    |     m3 = multiply_matrix(m2, m1)
    |     rxryrz1 = convert_matrix_to_axang(m3)
    |     rx1 = rxryrz1[0]
    |     ry1 = rxryrz1[1]
    |     rz1 = rxryrz1[2]
    | 
    |     point1 = p[p1x, p1y, p1z, rx1, ry1, rz1]
    | 
    |     # get second point (right) (point2)
    |     # take the center point and move right the radius plus the cushions
    |     p2x = pcx + vecrx * radius + vecrx * cusharound + vecnx * -1 * cushout
    |     p2y = pcy + vecry * radius + vecry * cusharound + vecny * -1 * cushout
    |     p2z = pcz
    | 
    |     # find rxryrz2
    |     # first rotation is 90 degrees about the x- axis
    |     m1 = get_rotation_matrix_from_description("x", -1, 90 * pi / 180)
    |     # second rotation is About 135 degrees about the z+ axis. This calculation is heading1 – 45 degrees
    |     m2 = get_rotation_matrix_from_description("z", 1, heading1 - 45 * pi/180)
    |     # combine them by multiplying
    |     m3 = multiply_matrix(m2, m1)
    |     rxryrz2 = convert_matrix_to_axang(m3)
    |     rx2 = rxryrz2[0]
    |     ry2 = rxryrz2[1]
    |     rz2 = rxryrz2[2]
    | 
    |     point2 = p[p2x, p2y, p2z, rx2, ry2, rz2]
    | 
    |     # get the third point (bottom) (point3)
    |     p3x = pcx + vecnx * -1 * cushout
    |     p3y = pcy + vecny * -1 * cushout
    |     p3z = pcz - vecuz * radius - vecuz * cusharound
    | 
    |     # find rxryrz3
    |     # first rotation is 45 degrees about the y+ axis
    |     m1 = get_rotation_matrix_from_description("y", 1, 45 * pi / 180)
    |     # second rotation is About 180 degrees about the z+ axis. This calculation is heading1 degrees
    |     m2 = get_rotation_matrix_from_description("z", 1, heading1)
    |     # combine them by multiplying
    |     m3 = multiply_matrix(m2, m1)
    |     rxryrz3 = convert_matrix_to_axang(m3)
    |     rx3 = rxryrz3[0]
    |     ry3 = rxryrz3[1]
    |     rz3 = rxryrz3[2]
    | 
    |     point3 = p[p3x, p3y, p3z, rx3, ry3, rz3]
    | 
    |     # get the fourth point (left) (point4)
    |     p4x = pcx - vecrx * radius - vecrx * cusharound + vecnx * -1 * cushout
    |     p4y = pcy - vecry * radius - vecry * cusharound + vecny * -1 * cushout
    |     p4z = pcz
    | 
    |     # find rxryrz4
    |     # first rotation is 90 degrees about the x+ axis
    |     m1 = get_rotation_matrix_from_description("x", 1, 90 * pi / 180)
    |     # second rotation is heading1 + 45 degrees about the z+ axis. approx 225 degrees ccw
    |     m2 = get_rotation_matrix_from_description("z", 1, heading1 + 45 * pi/180)
    |     # combine them by multiplying
    |     m3 = multiply_matrix(m2, m1)
    |     rxryrz4 = convert_matrix_to_axang(m3)
    |     rx4 = rxryrz4[0]
    |     ry4 = rxryrz4[1]
    |     rz4 = rxryrz4[2]
    | 
    |     point4 = p[p4x, p4y, p4z, rx4, ry4, rz4]
    | 
    |     # return the points
    |     ret = struct(point1=point1, point2=point2, point3=point3, point4=point4)
    |     return ret
    | 
    | end
    | 
    | # this function calculates the points necessary for the fillet sleeve weld path.
    | # this assumes a vertical plane
    | def calculate_points_sleeve_fillet(struct1):
    |     # get the stuff from the struct
    |     pcenter = struct1[0]
    |     pcx = pcenter[0]
    |     pcy = pcenter[1]
    |     pcz = pcenter[2]
    |     planenormalvec = struct1[1]
    |     radius = struct1[2]
    |     heading1 = struct1[3]
    |     vecn = struct1[4]
    |     vecnx = vecn[0]
    |     vecny = vecn[1]
    |     vecr = struct1[5]
    |     vecrx = vecr[0]
    |     vecry = vecr[1]
    |     vecu = struct1[6]
    |     vecuz = vecu[2]
    | 
    |     # define cushions (the backofhole can't actually touch the intersection of pipe and wall, it travels a certain distance around it
    |     cushout = 0.006 # 5mm # the cushion out from the wall
    |     cusharound = 0.004 # 5mm # the cushion around the sleeve.
    | 
    |     # get the top point (point1)
    |     # take the center point and move up the radius plus the cushions
    |     p1x = pcx + vecnx * -1 * cushout
    |     p1y = pcy + vecny * -1 * cushout
    |     p1z = pcz + vecuz * radius + vecuz * cusharound
    | 
    |     # find rxryrz1
    |     # first rotation is 135 degrees about the y- direction. 90 degrees to get flat. Tip pointing x-, preheat pointing y+. 45 more degrees to get at that above angle
    |     m1 = get_rotation_matrix_from_description("y", -1, 135 * pi / 180)
    |     # second rotation is heading1 – 180 degrees about the z+ axis to get pointing straight into wall. Heading1 should be about 180 degrees
    |     m2 = get_rotation_matrix_from_description("z", 1, heading1 - 180 * pi/180)
    |     # combine them by multiplying
    |     m3 = multiply_matrix(m2, m1)
    |     rxryrz1 = convert_matrix_to_axang(m3)
    |     rx1 = rxryrz1[0]
    |     ry1 = rxryrz1[1]
    |     rz1 = rxryrz1[2]
    | 
    |     point1 = p[p1x, p1y, p1z, rx1, ry1, rz1]
    | 
    |     # get second point (right) (point2)
    |     # take the center point and move right the radius plus the cushions
    |     p2x = pcx + vecrx * radius + vecrx * cusharound + vecnx * -1 * cushout
    |     p2y = pcy + vecry * radius + vecry * cusharound + vecny * -1 * cushout
    |     p2z = pcz
    | 
    |     # find rxryrz2
    |     # first rotation is 90 degrees about the x- axis
    |     m1 = get_rotation_matrix_from_description("x", -1, 90 * pi / 180)
    |     # second rotation is About 135 degrees about the z+ axis. This calculation is heading1 – 45 degrees
    |     m2 = get_rotation_matrix_from_description("z", 1, heading1 - 45 * pi/180)
    |     # combine them by multiplying
    |     m3 = multiply_matrix(m2, m1)
    |     rxryrz2 = convert_matrix_to_axang(m3)
    |     rx2 = rxryrz2[0]
    |     ry2 = rxryrz2[1]
    |     rz2 = rxryrz2[2]
    | 
    |     point2 = p[p2x, p2y, p2z, rx2, ry2, rz2]
    | 
    |     # get the third point (bottom) (point3)
    |     p3x = pcx + vecnx * -1 * cushout
    |     p3y = pcy + vecny * -1 * cushout
    |     p3z = pcz - vecuz * radius - vecuz * cusharound
    | 
    |     # find rxryrz3
    |     # first rotation is 45 degrees about the y+ axis
    |     m1 = get_rotation_matrix_from_description("y", 1, 45 * pi / 180)
    |     # second rotation is About 180 degrees about the z+ axis. This calculation is heading1 degrees
    |     m2 = get_rotation_matrix_from_description("z", 1, heading1)
    |     # combine them by multiplying
    |     m3 = multiply_matrix(m2, m1)
    |     rxryrz3 = convert_matrix_to_axang(m3)
    |     rx3 = rxryrz3[0]
    |     ry3 = rxryrz3[1]
    |     rz3 = rxryrz3[2]
    | 
    |     point3 = p[p3x, p3y, p3z, rx3, ry3, rz3]
    | 
    |     # get the fourth point (left) (point4)
    |     p4x = pcx - vecrx * radius - vecrx * cusharound + vecnx * -1 * cushout
    |     p4y = pcy - vecry * radius - vecry * cusharound + vecny * -1 * cushout
    |     p4z = pcz
    | 
    |     # find rxryrz4
    |     # first rotation is 90 degrees about the x+ axis
    |     m1 = get_rotation_matrix_from_description("x", 1, 90 * pi / 180)
    |     # second rotation is heading1 + 45 degrees about the z+ axis. approx 225 degrees ccw
    |     m2 = get_rotation_matrix_from_description("z", 1, heading1 + 45 * pi/180)
    |     # combine them by multiplying
    |     m3 = multiply_matrix(m2, m1)
    |     rxryrz4 = convert_matrix_to_axang(m3)
    |     rx4 = rxryrz4[0]
    |     ry4 = rxryrz4[1]
    |     rz4 = rxryrz4[2]
    | 
    |     point4 = p[p4x, p4y, p4z, rx4, ry4, rz4]
    | 
    |     # get the angle for the tilt-back at the top (p1)
    |     m0 = get_rotation_matrix_from_description("x", -1, 10 * pi / 180)
    |     m1 = get_rotation_matrix_from_description("y", -1, 135 * pi / 180)
    |     # second rotation is heading1 – 180 degrees about the z+ axis to get pointing straight into wall. Heading1 should be about 180 degrees
    |     m2 = get_rotation_matrix_from_description("z", 1, heading1 - 180 * pi/180)
    |     # combine them by multiplying
    |     m3 = multiply_matrix(m2, m1)
    |     m4 = multiply_matrix(m3, m0)
    |     rxryrz1tilt = convert_matrix_to_axang(m4)
    |     rx1t = rxryrz1tilt[0]
    |     ry1t = rxryrz1tilt[1]
    |     rz1t = rxryrz1tilt[2]
    | 
    |     # point 1, but with the tilt back angle
    |     point1t = p[p1x, p1y, p1z, rx1t, ry1t, rz1t]
    | 
    |     # point45 (the point 45 degrees along the path) (has no rxryrz data) (because if we do fixed angle circle move it wont use that anyways, it'l just use the angle from p1t)
    |     distup = cos(45 * pi/180) * (radius + cusharound)
    |     distover = sin(45 * pi/180) * (radius + cusharound)
    |     p45x = pcx + vecrx * distover + vecnx * -1 * cushout
    |     p45y = pcy + vecry * distover + vecny * -1 * cushout
    |     p45z = pcz + vecuz * distup
    |     point45 = p[p45x, p45y, p45z, 0,0,0]
    | 
    |     # point22 (22.5 degrees of angle)
    |     distup = cos(22.5 * pi/180) * (radius + cusharound)
    |     distover = sin(22.5 * pi/180) * (radius + cusharound)
    |     p22x = pcx + vecrx * distover + vecnx * -1 * cushout
    |     p22y = pcy + vecry * distover + vecny * -1 * cushout
    |     p22z = pcz + vecuz * distup
    |     point22 = p[p22x, p22y, p22z, 0,0,0]
    | 
    |     # return the points
    |     ret = struct(point1=point1, point2=point2, point3=point3, point4=point4, point1t=point1t, point45=point45, point22=point22)
    |     return ret
    | 
    | end
    | 
    | def make_pose_list(length):
    |     if length < 1:
    |         ret = []
    |         return ret
    |     end
    |     if length == 1:
    |         pose_list = [p[0, 0, 0, 0, 0, 0]]
    |         return pose_list
    |     end
    |     if length == 2:
    |         pose_list = [p[0, 0, 0, 0, 0, 0], p[0, 0, 0, 0, 0, 0]]
    |         return pose_list
    |     end
    |     if length == 3:
    |         pose_list = [p[0, 0, 0, 0, 0, 0], p[0, 0, 0, 0, 0, 0], p[0, 0, 0, 0, 0, 0]]
    |         return pose_list
    |     end
    |     if length == 4:
    |         pose_list = [p[0, 0, 0, 0, 0, 0], p[0, 0, 0, 0, 0, 0], p[0, 0, 0, 0, 0, 0], p[0, 0, 0, 0, 0, 0]]
    |         return pose_list
    |     end
    |     if length == 5:
    |         pose_list = [p[0, 0, 0, 0, 0, 0], p[0, 0, 0, 0, 0, 0], p[0, 0, 0, 0, 0, 0], p[0, 0, 0, 0, 0, 0], p[0, 0, 0, 0, 0, 0]]
    |         return pose_list
    |     end
    |     if length == 6:
    |         pose_list = [p[0, 0, 0, 0, 0, 0], p[0, 0, 0, 0, 0, 0], p[0, 0, 0, 0, 0, 0], p[0, 0, 0, 0, 0, 0], p[0, 0, 0, 0, 0, 0], p[0, 0, 0, 0, 0, 0]]
    |         return pose_list
    |     end
    |     if length == 7:
    |         pose_list = [p[0, 0, 0, 0, 0, 0], p[0, 0, 0, 0, 0, 0], p[0, 0, 0, 0, 0, 0], p[0, 0, 0, 0, 0, 0], p[0, 0, 0, 0, 0, 0], p[0, 0, 0, 0, 0, 0], p[0, 0, 0, 0, 0, 0]]
    |         return pose_list
    |     end
    |     if length == 8:
    |         pose_list = [p[0, 0, 0, 0, 0, 0], p[0, 0, 0, 0, 0, 0], p[0, 0, 0, 0, 0, 0], p[0, 0, 0, 0, 0, 0], p[0, 0, 0, 0, 0, 0], p[0, 0, 0, 0, 0, 0], p[0, 0, 0, 0, 0, 0], p[0, 0, 0, 0, 0, 0]]
    |         return pose_list
    |     end
    |     if length == 9:
    |         pose_list = [p[0, 0, 0, 0, 0, 0], p[0, 0, 0, 0, 0, 0], p[0, 0, 0, 0, 0, 0], p[0, 0, 0, 0, 0, 0], p[0, 0, 0, 0, 0, 0], p[0, 0, 0, 0, 0, 0], p[0, 0, 0, 0, 0, 0], p[0, 0, 0, 0, 0, 0], p[0, 0, 0, 0, 0, 0]]
    |         return pose_list
    |     end
    |     if length > 9:
    |         popuptext = "Program is only capable of storing 9 pegs at once. You selected more than 9. "
    |         # infinite loop
    |         while 1==1:
    |             popup(popuptext, title="Too Many Pegs",blocking=True)
    |         end
    |     end
    | end
    | 
    | # this function calculates the poses required on the weldpath for a specific teach pose for peg center.
    | # call this function for every peg you want to weld.
    | def main_calculate_peg(pose1):
    |     # constants
    |     peg_width = 2.05 # inches
    |     fixture_height = 1.5 # inches
    |     cushout = 0.006 # 5mm # the cushion out from the wall
    |     cusharound = 0.004 # 5mm # the cushion around the sleeve.
    |     delz = fixture_height *25.4/1000 - cushout
    |     rad = peg_width *1/2 * 25.4/1000 + cusharound
    | 
    |     # calculate angles
    |     # rxryrz1 (for point 1 (back side of peg)
    |     # start with gun facing up, shield tip pointing in x+ direction
    |     # rotate about y axis (y-) 135 degrees.
    |     # thats it. (for the other ones, then rotate 90 degrees about z axis from this spot
    |     m0 = get_rotation_matrix_from_description("y", -1, 225 * pi / 180)
    |     rxryrz1 = convert_matrix_to_axang(m0)
    |     rx1 = rxryrz1[0]
    |     ry1 = rxryrz1[1]
    |     rz1 = rxryrz1[2]
    | 
    |     # rxryrz2
    |     # second rotation is 90 degrees about z- axis
    |     m1 = get_rotation_matrix_from_description("z", -1, 90 * pi / 180)
    |     m2 = multiply_matrix(m1, m0)
    |     rxryrz2 = convert_matrix_to_axang(m2)
    |     rx2 = rxryrz2[0]
    |     ry2 = rxryrz2[1]
    |     rz2 = rxryrz2[2]
    | 
    |     # rxryrz3
    |     # second rotation is 180 degrees about z- axis
    |     m1 = get_rotation_matrix_from_description("z", -1, 180 * pi / 180)
    |     m2 = multiply_matrix(m1, m0)
    |     rxryrz3 = convert_matrix_to_axang(m2)
    |     rx3 = rxryrz3[0]
    |     ry3 = rxryrz3[1]
    |     rz3 = rxryrz3[2]
    | 
    |     # rxryrz4
    |     # second rotation is 270 degrees about z- axis
    |     m1 = get_rotation_matrix_from_description("z", -1, 270 * pi / 180)
    |     m2 = multiply_matrix(m1, m0)
    |     rxryrz4 = convert_matrix_to_axang(m2)
    |     rx4 = rxryrz4[0]
    |     ry4 = rxryrz4[1]
    |     rz4 = rxryrz4[2]
    | 
    |     # get points
    |     # get lift column height based on z value
    |     # if z is between +1 feet and -1 feet then go to 750
    |     # if z is greater than +1 feet but less than +4 feet, then go to 880
    |     # if z is greater than +4 feet, then error
    |     # if z is less than -1 feet, then go to 750 mm above z.
    | 
    |     # scrap that. new rules
    |     # go to 750 mm above z.
    |     # if that result is above 880, then go to 880.
    |     # that will work until we get problems
    | 
    |     z0 = pose1[2] # the teach point's z value (taken when lift column = 0)
    |     lczn = z0 + .750 # lift column z needed
    |     if lczn > .880:
    |         lczn = .880
    |     end
    |     liftcolumnzneeded = lczn * 1000 # set the z position
    |     zposerel = z0 - lczn # z pose relative = the teach point's z value at the new lift column position.
    | 
    |     pcenterx = pose1[0]
    |     pcentery = pose1[1]
    | 
    |     #points
    |     p1x = pcenterx - rad
    |     p1y = pcentery
    |     p1z = zposerel - delz
    | 
    |     p2x = pcenterx
    |     p2y = pcentery + rad
    |     p2z = zposerel - delz
    | 
    |     p3x = pcenterx + rad
    |     p3y = pcentery
    |     p3z = zposerel - delz
    | 
    |     p4x = pcenterx
    |     p4y = pcentery - rad
    |     p4z = zposerel - delz
    | 
    |     point1 = p[p1x, p1y, p1z, rx1, ry1, rz1]
    |     point2 = p[p2x, p2y, p2z, rx2, ry2, rz2]
    |     point3 = p[p3x, p3y, p3z, rx3, ry3, rz3]
    |     point4 = p[p4x, p4y, p4z, rx4, ry4, rz4]
    | 
    |     ret = struct(point1=point1, point2=point2, point3=point3, point4=point4, liftcolumnzneeded=liftcolumnzneeded)
    |     return ret
    | 
    | 
    | 
    | end
  SuppressedNode
    Script: welder_state_ready()
  SuppressedNode
    sidewallchoice :=  (valueSource=Operator message=Is the sidewall 3/4 inch? valueType=Boolean)
  SuppressedNode
    If sidewallchoice removedSiblings(If(type=Else checkContinuously=false, children(Assignment(valueSource=Expression, variable(name=sidewall), expression=0.375))))
      sidewall := 0.628
  SuppressedNode
    deepcham :=  (valueSource=Operator message=Is the chamfer extra deep? (more than 0.21) valueType=Boolean)
  SuppressedNode
    MoveJ speed 60 deg/s, acceleration 80 deg/s^2 (useActiveTCP=true optimoveEnabled=false optiMoveSpeed=0.3 optiMoveAcceleration=0.09) feature=Base
      Waypoint Waypoint_46: TCP in base x=894.108 y=351.078 z=354.456 mm, rx=2.3264 ry=2.0525 rz=0.0574 rad; joints [-187.182, -67.294, 94.726, 57.522, -0.141, -88.018] deg; TCP offset x=-5.49 y=-328 z=106.39 mm, rx=1.2092 ry=-1.2092 rz=1.2092 rad
  Set NoAction tcp=pretend_w_top
  Script: Test_Teach_Peg()
  Set NoAction tcp=pretend_w_top
  Script: kill threadId_Thread_1
  SuppressedNode
    Script: Cover_LT_Homing()
  MoveL speed 250 mm/s, acceleration 1200 mm/s^2 (useActiveTCP=true optimoveEnabled=false optiMoveSpeed=0.3 optiMoveAcceleration=0.09) feature=Base
    MoveDirectionNode (selectedDirection=ZPlus)
      Until DISTANCE (allowActions=false deceleration=3 distanceNodeType=STOP) Distance=0.1; motionParameters(blendRadius=0)
  MoveJ speed 60 deg/s, acceleration 80 deg/s^2 (useActiveTCP=true optimoveEnabled=false optiMoveSpeed=0.3 optiMoveAcceleration=0.09) feature=Base
    Waypoint Waypoint_3: TCP in base x=-565.561 y=-88.282 z=748.934 mm, rx=0.347 ry=3.1015 rz=-0.0385 rad; joints [-12.028, -113.359, 121.362, 263.351, -88.693, -89.284] deg; TCP offset x=0 y=0 z=19 mm, rx=0 ry=0 rz=0 rad
    Waypoint Waypoint_40: TCP in base x=360.688 y=270.12 z=646.145 mm, rx=0.0578 ry=2.126 rz=2.1341 rad; joints [-198.126, -117.852, 133.303, -13.01, -11.422, -6.036] deg
  Set NoAction tcp=pretend_welder
  Folder extrude knife
    lch := get_lift_column_height_condensed()
    If lch > 1
      URCap MachineLogic for Universal Robots (MachineLogic for Universal Robots, Vention Inc.) dataModel(type=addMotor, numberAdded=0, speed_in_mm_per_min=3000.0, acceleration_in_mm_per_s2=50.0, teachColor=BLUE, combo1=MachineMotion1, combo2=(1) Custom Actuator, combo3=Home, combo6=In series, message=Homing, description=Moves the actuator in the negative direction until the home sensor is triggered and sets position to zero (0)., comboAddress=Address 1, comboActuator=Valve 1)
      Script: extrude_knife3()
      URCap MachineLogic for Universal Robots (MachineLogic for Universal Robots, Vention Inc.) dataModel(type=addMotor, numberAdded=0, speed_in_mm_per_min=3000.0, acceleration_in_mm_per_s2=50.0, ActuatorPos=lch, teachColor=BLUE, combo1=MachineMotion1, combo2=(1) Custom Actuator, combo3=Move to Position, combo6=In series, message=Move to Position, description=Moves the actuator to a specified position from the home location., comboAddress=Address 1, comboActuator=Valve 1)
    Else 
      Script: extrude_knife3()
  dummy := main_calculate_peg(poses_list[0])
  Script: align_peg()
  pose_index := 0
  Loop While (checkContinuously=false) expression=pose_index < num_pegs
    Script: peg_unwind()
    pose_cur := poses_list[pose_index]
    pathturn := main_calculate_peg(pose_cur)
    Folder liftcolumnup
      liftcolumnz := liftcolumnzneeded
      URCap MachineLogic for Universal Robots (MachineLogic for Universal Robots, Vention Inc.) dataModel(type=addMotor, numberAdded=0, acceleration_in_mm_per_s2=50.0, ActuatorPos=liftcolumnz, speed_in_mm_per_min=6000.0, teachColor=BLUE, combo1=MachineMotion1, combo2=(1) Custom Actuator, combo3=Move to Position, combo6=In series, message=Move to Position, description=Moves the actuator to a specified position from the home location., comboAddress=Address 1, comboActuator=Valve 1)
    Script: weld_peg()
    pose_index := pose_index +1
  SuppressedNode
    pathturn := main_calculate_pegs(poses_list)
  SuppressedNode
    Script: move_path_cover_lt()
  Set NoAction tcp=pretend_welder
  MoveJ speed 60 deg/s, acceleration 80 deg/s^2 (useActiveTCP=true optimoveEnabled=false optiMoveSpeed=0.3 optiMoveAcceleration=0.09) feature=Base
    Waypoint Waypoint_8: TCP in base x=-262.599 y=-117.911 z=443.767 mm, rx=0.1153 ry=3.1146 rz=0.2657 rad; joints [5.497, -142.032, 129.309, 13.11, 99.793, -9.621] deg; TCP offset x=-9.5 y=-328 z=105.73 mm, rx=1.2092 ry=-1.2092 rz=1.2092 rad
    Waypoint Waypoint_9: TCP in base x=397.354 y=356.263 z=319.809 mm, rx=2.3163 ry=2.0576 rz=0.0741 rad; joints [-198.308, -118.162, 133.452, -12.561, -11.517, -6.326] deg
  URCap MachineLogic for Universal Robots (MachineLogic for Universal Robots, Vention Inc.) dataModel(type=addMotor, numberAdded=0, speed_in_mm_per_min=3000.0, acceleration_in_mm_per_s2=50.0, teachColor=BLUE, combo1=MachineMotion1, combo2=(1) Custom Actuator, combo3=Home, combo6=In series, message=Homing, description=Moves the actuator in the negative direction until the home sensor is triggered and sets position to zero (0)., comboAddress=Address 1, comboActuator=Valve 1)
  SafeHome (positionOptionType=SPEED_AND_ACCELERATION speed=1.047198 acceleration=1.396263 nextMotionTime=2)
SubProgram Test_Teach_Peg (keepSynchronizedWithDisk=false) programFile=/programs/Test Teach Peg.urp
  Set NoAction tcp=pretend_w_top
  SuppressedNode
    MoveL speed 250 mm/s, acceleration 1200 mm/s^2 (useActiveTCP=true optimoveEnabled=false optiMoveSpeed=0.3 optiMoveAcceleration=0.09) feature=Base
      Waypoint Waypoint_1: TCP in base x=183.613 y=373.491 z=464.002 mm, rx=0 ry=3.1416 rz=0 rad; joints [-144.817, -120.486, 148.461, -117.931, -90.033, 125.101] deg; TCP offset x=0 y=0 z=19 mm, rx=0 ry=0 rz=0 rad
      'move welder up out of holder'
  Folder ask how many
    num_pegs :=  (valueSource=Operator message=Weld how many pegs now? valueType=Integer)
    If num_pegs<1
      Loop Forever
        Popup Message (haltProgram=false message=invalid: negative number given. restart program inputType=Text)
    poses_list := make_pose_list(num_pegs)
    pose_index := 0
  MoveJ speed 60 deg/s, acceleration 80 deg/s^2 (useActiveTCP=false optimoveEnabled=false optiMoveSpeed=0.3 optiMoveAcceleration=0.09) tcp=TCP_1_plate; feature=Base
    Waypoint Waypoint_40: TCP in base x=360.688 y=270.12 z=646.145 mm, rx=0.0578 ry=2.126 rz=2.1341 rad; joints [-198.126, -117.852, 133.303, -13.01, -11.422, -6.036] deg
    'above waypoint is home'
    SuppressedNode
      Waypoint Waypoint_2: TCP in base x=-548.957 y=386.285 z=143.71 mm, rx=1.5708 ry=0 rz=0 rad; joints [-60.253, -57.926, 123.544, -65.529, -60.311, -0.099] deg
    Waypoint Waypoint_3: TCP in base x=-565.561 y=-88.282 z=748.934 mm, rx=0.347 ry=3.1015 rz=-0.0385 rad; joints [-12.028, -113.359, 121.362, 263.351, -88.693, -89.284] deg
  Set NoAction tcp=pretend_w_top
  freedrive_m_var := False
  freedrive_m_var := True
  Loop While (checkContinuously=false) expression=pose_index < num_pegs
    Popup Message (haltProgram=false message=Move the TCP to the peg fixture center, then click 'Continue' inputType=Text)
    tcp_pose_left := get_actual_tcp_pose()
    Script: poses_list[pose_index] = tcp_pose_left
    Wait Sleep waitTime=1
    pose_index := pose_index +1
  SuppressedNode
    Popup Message (haltProgram=false message=Move the TCP to the right side of the weld (very center of groove), then click 'Continue' inputType=Text)
  SuppressedNode
    tcp_pose_right := get_actual_tcp_pose()
  freedrive_m_var := False
  Wait Sleep waitTime=0.25
  Script: sync()
SubProgram weld_peg (keepSynchronizedWithDisk=false)
  Set NoAction tcp=sleeve_piv
  'get the points'
  p1 := pathturn[0]
  p2 := pathturn[1]
  p3 := pathturn[2]
  p4 := pathturn[3]
  p1a1 := p[p1[0]-0.02,p1[1],p1[2]+0.05,p1[3],p1[4],p1[5]]
  'assume its already aligned somewhat over the tank area'
  MoveL speed 100 mm/s, acceleration 1200 mm/s^2 (useActiveTCP=true optimoveEnabled=false optiMoveSpeed=0.3 optiMoveAcceleration=0.09) feature=Base
    Waypoint Variable (Variable): variable=p1a1
  MoveL speed 10 mm/s, acceleration 1200 mm/s^2 (useActiveTCP=true optimoveEnabled=false optiMoveSpeed=0.3 optiMoveAcceleration=0.09) feature=Base
    Waypoint Variable (Variable): variable=p1
  'preheat'
  Wait Sleep waitTime=6
  'turn extrusion on'
  URCap WireTank Serial (WireTank Serial, WireTank, LLC) dataModel(NODE_TITLE=Serial Bridge uR1, Command=[252,82,49], QUERY=false, byte_array=true, OUTPUT_ENTRY=Static, Variable(key=OUTPUT_VARIABLE, variable(name=HwResp)))
  Wait Sleep waitTime=1.2
  Set DigitalOutput pin=digital_out[0]; digitalValue=1
  MoveP speed 10 mm/s, acceleration 1200 mm/s^2 (blendRadius=0.025 useActiveTCP=true optimoveEnabled=false optiMoveSpeed=0.3 optiMoveAcceleration=0.09) feature=Base
    CircleMove (OrientationMode=FIXED)
      Waypoint Variable (Variable): variable=p2
      Waypoint Variable (Variable): variable=p3
    CircleMove (OrientationMode=FIXED)
      Waypoint Variable (Variable): variable=p4
      Waypoint Variable (Variable): variable=p1
  'turn extrusion off'
  URCap WireTank Serial (WireTank Serial, WireTank, LLC) dataModel(QUERY=false, NODE_TITLE=Serial Bridge uR0, Command=[252,82,48], byte_array=true, OUTPUT_ENTRY=Static, Variable(key=OUTPUT_VARIABLE, variable=HwResp))
  MoveP speed 10 mm/s, acceleration 1200 mm/s^2 (blendRadius=0.025 useActiveTCP=true optimoveEnabled=false optiMoveSpeed=0.3 optiMoveAcceleration=0.09) feature=Base
    CircleMove (OrientationMode=FIXED)
      Waypoint Variable (Variable): variable=p2
      Waypoint Variable (Variable): variable=p3
  Set DigitalOutput pin=digital_out[0]; digitalValue=0
  'retreat'
  MoveL speed 250 mm/s, acceleration 1200 mm/s^2 (useActiveTCP=true optimoveEnabled=false optiMoveSpeed=0.3 optiMoveAcceleration=0.09) feature=Base
    MoveDirectionNode (selectedDirection=ZPlus)
      Until DISTANCE (allowActions=false deceleration=3 distanceNodeType=STOP) Distance=0.1; motionParameters(blendRadius=0)
SubProgram align_peg (keepSynchronizedWithDisk=false) programFile=/programs/align_peg.urp
  'leave home'
  SuppressedNode
    Set NoAction tcp=pretend_welder
  SuppressedNode
    URCap MachineLogic for Universal Robots (MachineLogic for Universal Robots, Vention Inc.) dataModel(type=addMotor, numberAdded=0, speed_in_mm_per_min=3000.0, acceleration_in_mm_per_s2=50.0, ActuatorPos=liftcolumnzneeded, teachColor=BLUE, combo1=MachineMotion1, combo2=(1) Custom Actuator, combo3=Move to Position, combo6=In series, message=Move to Position, description=Moves the actuator to a specified position from the home location., comboAddress=Address 1, comboActuator=Valve 1)
  Folder liftcolumnup
    liftcolumnz := liftcolumnzneeded
    URCap MachineLogic for Universal Robots (MachineLogic for Universal Robots, Vention Inc.) dataModel(type=addMotor, numberAdded=0, acceleration_in_mm_per_s2=50.0, ActuatorPos=liftcolumnz, teachColor=BLUE, combo1=MachineMotion1, combo2=(1) Custom Actuator, combo3=Move to Position, combo6=In series, message=Move to Position, description=Moves the actuator to a specified position from the home location., comboAddress=Address 1, comboActuator=Valve 1, speed_in_mm_per_min=6000.0)
  SuppressedNode
    MoveJ speed 60 deg/s, acceleration 80 deg/s^2 (useActiveTCP=true optimoveEnabled=false optiMoveSpeed=0.3 optiMoveAcceleration=0.09) feature=Base
      Waypoint Waypoint_1: TCP in base x=439.488 y=377.651 z=439.882 mm, rx=2.2965 ry=2.0951 rz=-0.0644 rad; joints [-188.975, -96.657, 133.035, 103.058, 4.742, -139.298] deg; TCP offset x=-9.5 y=-328 z=105 mm, rx=1.2092 ry=-1.2092 rz=1.2092 rad
      Waypoint Waypoint_2: TCP in base x=-567.049 y=119.272 z=439.882 mm, rx=-0.8568 ry=2.9689 rz=0.0164 rad; joints [-61.526, -96.657, 133.035, 103.058, 4.742, -139.298] deg
  'spin?'
  'points'
  SuppressedNode
    If 1≟2
      'tilt'
      MoveJ speed 60 deg/s, acceleration 80 deg/s^2 (useActiveTCP=true optimoveEnabled=false optiMoveSpeed=0.3 optiMoveAcceleration=0.09) feature=Base
        Waypoint Waypoint_3: TCP in base x=-782.323 y=119.272 z=439.882 mm, rx=-0.1409 ry=-2.6543 rz=-0.0579 rad; joints [-38.432, -118.572, 138.524, -52.025, 61.559, 15.606] deg
        Waypoint Waypoint_4: TCP in base x=-839.555 y=157.82 z=59.483 mm, rx=-0.1359 ry=-2.576 rz=-0.0621 rad; joints [-38.672, -71.334, 157.907, -123.561, 62.634, 17.978] deg
      MoveJ speed 60 deg/s, acceleration 80 deg/s^2 (useActiveTCP=true optimoveEnabled=false optiMoveSpeed=0.3 optiMoveAcceleration=0.09) feature=Base
        Waypoint Waypoint_5: TCP in base x=-839.555 y=157.82 z=154.033 mm, rx=-0.1359 ry=-2.576 rz=-0.0621 rad; joints [-38.663, -86.736, 154.954, -105.21, 62.654, 17.987] deg
        Waypoint Waypoint_6: TCP in base x=-930.504 y=247.449 z=154.033 mm, rx=1.7264 ry=-2.0251 rz=0.4813 rad; joints [-47.448, -44.223, 108.584, -199.171, 48.598, 145.286] deg
        Waypoint Waypoint_7: TCP in base x=-1008.947 y=181.992 z=154.033 mm, rx=2.8737 ry=-0.4936 rz=0.8267 rad; joints [-21.503, -27.525, 68.369, -188.611, 91.899, 180.193] deg
        Waypoint Waypoint_8: TCP in base x=-1005.76 y=182.333 z=166.844 mm, rx=2.9972 ry=-0.3869 rz=0.8133 rad; joints [-19.507, -27.075, 40.49, 16.635, -93.289, 5.373] deg
      MoveJ speed 60 deg/s, acceleration 80 deg/s^2 (useActiveTCP=true optimoveEnabled=false optiMoveSpeed=0.3 optiMoveAcceleration=0.09) feature=Base
        Waypoint Waypoint_9: TCP in base x=-1005.76 y=135.995 z=-301.87 mm, rx=-2.9509 ry=-0.1653 rz=-0.7853 rad; joints [-11.926, -9.754, 42.428, -1.512, -104.955, 12.357] deg
      'actual'
      MoveJ speed 60 deg/s, acceleration 80 deg/s^2 (useActiveTCP=true optimoveEnabled=false optiMoveSpeed=0.3 optiMoveAcceleration=0.09) feature=Base
        Waypoint Waypoint_13: TCP in base x=-820.615 y=235.067 z=-600.712 mm, rx=2.789 ry=-0.3984 rz=-1.1799 rad; joints [-36.349, -28.171, 124.415, -140.933, -100.235, -24.393] deg
        Waypoint Waypoint_12: TCP in base x=-1004.07 y=104.199 z=-600.712 mm, rx=-1.7423 ry=1.8799 rz=0.9101 rad; joints [-16.137, -21.262, 116.105, -178.633, -44.236, 66.954] deg
        Waypoint Waypoint_11: TCP in base x=-1004.07 y=251.363 z=-600.712 mm, rx=0.2287 ry=2.3379 rz=0.1546 rad; joints [-20.059, -11.78, 93.702, -217.985, -87.895, 163.36] deg
        Waypoint Waypoint_10: TCP in base x=-813.178 y=367.752 z=-600.712 mm, rx=1.8208 ry=1.595 rz=-0.5735 rad; joints [-36.866, -15.96, 106.588, -203.107, -131.508, 223.468] deg
  SuppressedNode
    If 1≟2
      Folder first try
        'worked pretty good. my 4 points were not a circle so it moved kind of wonky. but still spun'
        MoveJ speed 60 deg/s, acceleration 80 deg/s^2 (useActiveTCP=true optimoveEnabled=false optiMoveSpeed=0.3 optiMoveAcceleration=0.09) feature=Base
          Waypoint Waypoint_13: TCP in base x=-820.615 y=235.067 z=-600.712 mm, rx=2.789 ry=-0.3984 rz=-1.1799 rad; joints [-36.349, -28.171, 124.415, -140.933, -100.235, -24.393] deg
        MoveP speed 10 mm/s, acceleration 1200 mm/s^2 (blendRadius=0.025 useActiveTCP=true optimoveEnabled=false optiMoveSpeed=0.3 optiMoveAcceleration=0.09) feature=Base
          CircleMove (OrientationMode=FIXED)
            Waypoint Waypoint_12: TCP in base x=-1004.07 y=104.199 z=-600.712 mm, rx=-1.7423 ry=1.8799 rz=0.9101 rad; joints [-16.137, -21.262, 116.105, -178.633, -44.236, 66.954] deg
            Waypoint Waypoint_11: TCP in base x=-1004.07 y=251.363 z=-600.712 mm, rx=0.2287 ry=2.3379 rz=0.1546 rad; joints [-20.059, -11.78, 93.702, -217.985, -87.895, 163.36] deg
          CircleMove (OrientationMode=FIXED)
            Waypoint Waypoint_10: TCP in base x=-813.178 y=367.752 z=-600.712 mm, rx=1.8208 ry=1.595 rz=-0.5735 rad; joints [-36.866, -15.96, 106.588, -203.107, -131.508, 223.468] deg
            Waypoint Waypoint_13: TCP in base x=-820.615 y=235.067 z=-600.712 mm, rx=2.789 ry=-0.3984 rz=-1.1799 rad; joints [-36.349, -28.171, 124.415, -140.933, -100.235, -24.393] deg
  SuppressedNode
    Folder second try
      'worked pretty good. my 4 points were not a circle so it moved kind of wonky. but still spun'
      MoveJ speed 60 deg/s, acceleration 80 deg/s^2 (useActiveTCP=true optimoveEnabled=false optiMoveSpeed=0.3 optiMoveAcceleration=0.09) feature=Base
        Waypoint Waypoint_13: TCP in base x=-820.615 y=235.067 z=-600.712 mm, rx=2.789 ry=-0.3984 rz=-1.1799 rad; joints [-36.349, -28.171, 124.415, -140.933, -100.235, -24.393] deg
      MoveL speed 250 mm/s, acceleration 1200 mm/s^2 (useActiveTCP=true optimoveEnabled=false optiMoveSpeed=0.3 optiMoveAcceleration=0.09) feature=Base
        Waypoint Waypoint_14: TCP in base x=-933.006 y=247.304 z=-556.073 mm, rx=2.8803 ry=-0.0661 rz=-1.2302 rad; joints [-29.557, -31.673, 118.683, -136.217, -107.709, -21.437] deg
      MoveP speed 10 mm/s, acceleration 1200 mm/s^2 (blendRadius=0.025 useActiveTCP=true optimoveEnabled=false optiMoveSpeed=0.3 optiMoveAcceleration=0.09) feature=Base
        CircleMove (OrientationMode=FIXED)
          Waypoint ViaPoint_1: TCP in base x=-997.806 y=207.515 z=-556.073 mm, rx=-1.6876 ry=1.8024 rz=0.7466 rad; joints [-20.307, -26.743, 112.915, -161.612, -48.271, 66.703] deg
          Waypoint EndPoint_1: TCP in base x=-1049.868 y=270.629 z=-561.34 mm, rx=0.1326 ry=2.3308 rz=-0.0225 rad; joints [-23.206, -14.525, 91.047, -209.147, -79.208, 166.32] deg
        CircleMove (OrientationMode=FIXED)
          Waypoint ViaPoint_2: TCP in base x=-979.337 y=322.737 z=-561.34 mm, rx=1.8079 ry=1.682 rz=-0.747 rad; joints [-31.834, -18.679, 101.995, -196.68, -128.219, 232.931] deg
          Waypoint Waypoint_14: TCP in base x=-933.006 y=247.304 z=-556.073 mm, rx=2.8803 ry=-0.0661 rz=-1.2302 rad; joints [-29.557, -31.673, 118.683, -136.217, -107.709, -21.437] deg
        CircleMove (OrientationMode=FIXED)
          Waypoint ViaPoint_1: TCP in base x=-997.806 y=207.515 z=-556.073 mm, rx=-1.6876 ry=1.8024 rz=0.7466 rad; joints [-20.307, -26.743, 112.915, -161.612, -48.271, 66.703] deg
          Waypoint EndPoint_1: TCP in base x=-1049.868 y=270.629 z=-561.34 mm, rx=0.1326 ry=2.3308 rz=-0.0225 rad; joints [-23.206, -14.525, 91.047, -209.147, -79.208, 166.32] deg
  SuppressedNode
    Folder third try
      'worked pretty good. my 4 points were not a circle so it moved kind of wonky. but still spun'
      MoveJ speed 60 deg/s, acceleration 80 deg/s^2 (useActiveTCP=true optimoveEnabled=false optiMoveSpeed=0.3 optiMoveAcceleration=0.09) feature=Base
        Waypoint Waypoint_13: TCP in base x=-820.615 y=235.067 z=-600.712 mm, rx=2.789 ry=-0.3984 rz=-1.1799 rad; joints [-36.349, -28.171, 124.415, -140.933, -100.235, -24.393] deg
      MoveL speed 250 mm/s, acceleration 1200 mm/s^2 (useActiveTCP=true optimoveEnabled=false optiMoveSpeed=0.3 optiMoveAcceleration=0.09) feature=Base
        Waypoint Waypoint_14: TCP in base x=-933.006 y=247.304 z=-556.073 mm, rx=2.8803 ry=-0.0661 rz=-1.2302 rad; joints [-29.557, -31.673, 118.683, -136.217, -107.709, -21.437] deg
      MoveJ speed 60 deg/s, acceleration 80 deg/s^2 (useActiveTCP=true optimoveEnabled=false optiMoveSpeed=0.3 optiMoveAcceleration=0.09) feature=Base
        Waypoint Waypoint_15: TCP in base x=-1155.523 y=247.304 z=-556.073 mm, rx=0.1075 ry=2.332 rz=-0.0118 rad; joints [-20.182, -12.844, 81.619, -201.64, -80.424, -192.34] deg
      MoveL speed 250 mm/s, acceleration 1200 mm/s^2 (useActiveTCP=true optimoveEnabled=false optiMoveSpeed=0.3 optiMoveAcceleration=0.09) feature=Base
        Waypoint EndPoint_1: TCP in base x=-1049.868 y=270.629 z=-561.34 mm, rx=0.1326 ry=2.3308 rz=-0.0225 rad; joints [-23.206, -14.525, 91.047, -209.147, -79.208, 166.32] deg
      Wait Sleep waitTime=1
      MoveP speed 10 mm/s, acceleration 1200 mm/s^2 (blendRadius=0.025 useActiveTCP=true optimoveEnabled=false optiMoveSpeed=0.3 optiMoveAcceleration=0.09) feature=Base
        CircleMove (OrientationMode=FIXED)
          Waypoint ViaPoint_2: TCP in base x=-979.337 y=322.737 z=-561.34 mm, rx=1.8079 ry=1.682 rz=-0.747 rad; joints [-31.834, -18.679, 101.995, -196.68, -128.219, 232.931] deg
          Waypoint Waypoint_14: TCP in base x=-933.006 y=247.304 z=-556.073 mm, rx=2.8803 ry=-0.0661 rz=-1.2302 rad; joints [-29.557, -31.673, 118.683, -136.217, -107.709, -21.437] deg
        CircleMove (OrientationMode=FIXED)
          Waypoint ViaPoint_1: TCP in base x=-997.806 y=207.515 z=-556.073 mm, rx=-1.6876 ry=1.8024 rz=0.7466 rad; joints [-20.307, -26.743, 112.915, -161.612, -48.271, 66.703] deg
          Waypoint EndPoint_1: TCP in base x=-1049.868 y=270.629 z=-561.34 mm, rx=0.1326 ry=2.3308 rz=-0.0225 rad; joints [-23.206, -14.525, 91.047, -209.147, -79.208, 166.32] deg
        CircleMove (OrientationMode=FIXED)
          Waypoint ViaPoint_2: TCP in base x=-979.337 y=322.737 z=-561.34 mm, rx=1.8079 ry=1.682 rz=-0.747 rad; joints [-31.834, -18.679, 101.995, -196.68, -128.219, 232.931] deg
          Waypoint Waypoint_14: TCP in base x=-933.006 y=247.304 z=-556.073 mm, rx=2.8803 ry=-0.0661 rz=-1.2302 rad; joints [-29.557, -31.673, 118.683, -136.217, -107.709, -21.437] deg
  SuppressedNode
    Folder fourth (peg)
      'worked pretty good. my 4 points were not a circle so it moved kind of wonky. but still spun'
      MoveJ speed 60 deg/s, acceleration 80 deg/s^2 (useActiveTCP=true optimoveEnabled=false optiMoveSpeed=0.3 optiMoveAcceleration=0.09) feature=Base
        Waypoint Waypoint_13: TCP in base x=-820.615 y=235.067 z=-600.712 mm, rx=2.789 ry=-0.3984 rz=-1.1799 rad; joints [-36.349, -28.171, 124.415, -140.933, -100.235, -24.393] deg
      MoveL speed 250 mm/s, acceleration 1200 mm/s^2 (useActiveTCP=true optimoveEnabled=false optiMoveSpeed=0.3 optiMoveAcceleration=0.09) feature=Base
        Waypoint Waypoint_14: TCP in base x=-933.006 y=247.304 z=-556.073 mm, rx=2.8803 ry=-0.0661 rz=-1.2302 rad; joints [-29.557, -31.673, 118.683, -136.217, -107.709, -21.437] deg
      MoveJ speed 60 deg/s, acceleration 80 deg/s^2 (useActiveTCP=true optimoveEnabled=false optiMoveSpeed=0.3 optiMoveAcceleration=0.09) feature=Base
        Waypoint Waypoint_15: TCP in base x=-1155.523 y=247.304 z=-556.073 mm, rx=0.1075 ry=2.332 rz=-0.0118 rad; joints [-20.182, -12.844, 81.619, -201.64, -80.424, -192.34] deg
      MoveL speed 250 mm/s, acceleration 1200 mm/s^2 (useActiveTCP=true optimoveEnabled=false optiMoveSpeed=0.3 optiMoveAcceleration=0.09) feature=Base
        Waypoint Waypoint_17: TCP in base x=-941.011 y=247.304 z=-664.711 mm, rx=0.1107 ry=2.4446 rz=-0.0059 rad; joints [-25.301, -8.351, 98.215, -228.375, -75.252, -194.663] deg
        Waypoint Waypoint_16: TCP in base x=-941.011 y=247.304 z=-712.565 mm, rx=0.1107 ry=2.4446 rz=-0.0059 rad; joints [-25.303, -5.145, 95.455, -228.821, -75.25, -194.666] deg
      Wait Sleep waitTime=2
      MoveP speed 10 mm/s, acceleration 1200 mm/s^2 (blendRadius=0.025 useActiveTCP=true optimoveEnabled=false optiMoveSpeed=0.3 optiMoveAcceleration=0.09) feature=Base
        CircleMove (OrientationMode=FIXED)
          Waypoint ViaPoint_3: TCP in base x=-902.128 y=271.937 z=-712.565 mm, rx=1.8739 ry=1.7594 rz=-0.6531 rad; joints [-29.151, -8.204, 102.29, -210.895, -134.312, -127.809] deg
          Waypoint EndPoint_2: TCP in base x=-879.998 y=228.196 z=-712.565 mm, rx=-2.9313 ry=0.1903 rz=1.0627 rad; joints [-28.767, -21.46, 113.717, -133.842, -105.761, -15.36] deg
        CircleMove (OrientationMode=FIXED)
          Waypoint ViaPoint_4: TCP in base x=-916.094 y=204.675 z=-712.565 mm, rx=-1.7817 ry=1.8631 rz=0.6704 rad; joints [-24.822, -17.392, 113.115, -161.812, -44.424, 56.385] deg
          Waypoint Waypoint_16: TCP in base x=-941.011 y=247.304 z=-712.565 mm, rx=0.1107 ry=2.4446 rz=-0.0059 rad; joints [-25.303, -5.145, 95.455, -228.821, -75.25, -194.666] deg
        CircleMove (OrientationMode=FIXED)
          Waypoint ViaPoint_3: TCP in base x=-902.128 y=271.937 z=-712.565 mm, rx=1.8739 ry=1.7594 rz=-0.6531 rad; joints [-29.151, -8.204, 102.29, -210.895, -134.312, -127.809] deg
          Waypoint EndPoint_2: TCP in base x=-879.998 y=228.196 z=-712.565 mm, rx=-2.9313 ry=0.1903 rz=1.0627 rad; joints [-28.767, -21.46, 113.717, -133.842, -105.761, -15.36] deg
  Folder fifth (backofhole)
    'worked pretty good. my 4 points were not a circle so it moved kind of wonky. but still spun'
    Set NoAction tcp=backofhole
    MoveJ speed 60 deg/s, acceleration 80 deg/s^2 (useActiveTCP=true optimoveEnabled=false optiMoveSpeed=0.3 optiMoveAcceleration=0.09) feature=Base
      Waypoint Waypoint_1: TCP in base x=439.488 y=377.651 z=439.882 mm, rx=2.2965 ry=2.0951 rz=-0.0644 rad; joints [-188.975, -96.657, 133.035, 103.058, 4.742, -139.298] deg
      Waypoint Waypoint_4: TCP in base x=-567.049 y=119.272 z=439.882 mm, rx=-0.8568 ry=2.9689 rz=0.0164 rad; joints [-61.526, -96.657, 133.035, 103.058, 4.742, -139.298] deg
    MoveJ speed 60 deg/s, acceleration 80 deg/s^2 (useActiveTCP=true optimoveEnabled=false optiMoveSpeed=0.3 optiMoveAcceleration=0.09) feature=Base
      Waypoint Waypoint_13: TCP in base x=-820.615 y=235.067 z=-600.712 mm, rx=2.789 ry=-0.3984 rz=-1.1799 rad; joints [-36.349, -28.171, 124.415, -140.933, -100.235, -24.393] deg
    MoveL speed 250 mm/s, acceleration 1200 mm/s^2 (useActiveTCP=true optimoveEnabled=false optiMoveSpeed=0.3 optiMoveAcceleration=0.09) feature=Base
      Waypoint Waypoint_14: TCP in base x=-933.006 y=247.304 z=-556.073 mm, rx=2.8803 ry=-0.0661 rz=-1.2302 rad; joints [-29.557, -31.673, 118.683, -136.217, -107.709, -21.437] deg
    MoveJ speed 60 deg/s, acceleration 80 deg/s^2 (useActiveTCP=true optimoveEnabled=false optiMoveSpeed=0.3 optiMoveAcceleration=0.09) feature=Base
      Waypoint Waypoint_15: TCP in base x=-1155.523 y=247.304 z=-556.073 mm, rx=0.1075 ry=2.332 rz=-0.0118 rad; joints [-20.182, -12.844, 81.619, -201.64, -80.424, -192.34] deg
    'end of approach'
    SuppressedNode
      MoveL speed 250 mm/s, acceleration 1200 mm/s^2 (useActiveTCP=true optimoveEnabled=false optiMoveSpeed=0.3 optiMoveAcceleration=0.09) feature=Base
        Waypoint Waypoint_18: TCP in base x=-939.675 y=242.159 z=-688.931 mm, rx=0.1858 ry=2.4403 rz=-0.0331 rad; joints [-25.871, -6.691, 96.723, -229.022, -77.473, -192.661] deg; TCP offset x=4.51 y=-328 z=105 mm, rx=1.2092 ry=-1.2092 rz=1.2092 rad
        Waypoint Waypoint_19: TCP in base x=-939.675 y=242.159 z=-719.896 mm, rx=0.1858 ry=2.4403 rz=-0.0331 rad; joints [-25.872, -4.62, 94.895, -229.263, -77.472, -192.663] deg
    SuppressedNode
      Wait Sleep waitTime=2
    SuppressedNode
      MoveP speed 10 mm/s, acceleration 1200 mm/s^2 (blendRadius=0.025 useActiveTCP=true optimoveEnabled=false optiMoveSpeed=0.3 optiMoveAcceleration=0.09) feature=Base
        CircleMove (OrientationMode=FIXED)
          Waypoint ViaPoint_5: TCP in base x=-907.205 y=264.785 z=-719.9 mm, rx=1.8738 ry=1.7594 rz=-0.6531 rad; joints [-28.993, -7.691, 102.75, -211.731, -134.382, -127.614] deg
          Waypoint EndPoint_3: TCP in base x=-881.393 y=236.092 z=-719.9 mm, rx=-2.9216 ry=0.2235 rz=1.0597 rad; joints [-28.315, -21.001, 113.308, -133.575, -104.432, -14.143] deg
        CircleMove (OrientationMode=FIXED)
          Waypoint ViaPoint_6: TCP in base x=-912.548 y=210.58 z=-719.9 mm, rx=-1.7177 ry=1.9091 rz=0.6478 rad; joints [-24.877, -16.344, 111.718, -164.775, -43.133, 60.968] deg
          Waypoint Waypoint_19: TCP in base x=-939.675 y=242.159 z=-719.896 mm, rx=0.1858 ry=2.4403 rz=-0.0331 rad; joints [-25.872, -4.62, 94.895, -229.263, -77.472, -192.663] deg
        CircleMove (OrientationMode=FIXED)
          Waypoint ViaPoint_5: TCP in base x=-907.205 y=264.785 z=-719.9 mm, rx=1.8738 ry=1.7594 rz=-0.6531 rad; joints [-28.993, -7.691, 102.75, -211.731, -134.382, -127.614] deg
          Waypoint EndPoint_3: TCP in base x=-881.393 y=236.092 z=-719.9 mm, rx=-2.9216 ry=0.2235 rz=1.0597 rad; joints [-28.315, -21.001, 113.308, -133.575, -104.432, -14.143] deg
SubProgram peg_unwind (keepSynchronizedWithDisk=false) programFile=/programs/peg_unwind.urp
  SuppressedNode
    MoveJ speed 60 deg/s, acceleration 80 deg/s^2 (useActiveTCP=true optimoveEnabled=false optiMoveSpeed=0.3 optiMoveAcceleration=0.09) feature=Base
      Waypoint start_pos: TCP in base x=-895.951 y=163.612 z=-688.729 mm, rx=-2.705 ry=0.5717 rz=1.1205 rad; joints [-22.749, -22.348, 117.732, -140.343, -89.229, 360.823] deg
      Waypoint Waypoint_2: TCP in base x=-855.562 y=110.096 z=-683.965 mm, rx=2.765 ry=-0.0879 rz=-1.1876 rad; joints [-26.005, -21.395, 121.77, -147.517, -102.002, 335.571] deg
  SuppressedNode
    Folder fifth (backofhole)
      'worked pretty good. my 4 points were not a circle so it moved kind of wonky. but still spun'
      Set NoAction tcp=backofhole
      MoveJ speed 60 deg/s, acceleration 80 deg/s^2 (useActiveTCP=true optimoveEnabled=false optiMoveSpeed=0.3 optiMoveAcceleration=0.09) feature=Base
        SuppressedNode
          Waypoint Waypoint_1: 
        Waypoint Waypoint_4: TCP in base x=-567.049 y=119.272 z=439.882 mm, rx=-0.8568 ry=2.9689 rz=0.0164 rad; joints [-61.526, -96.657, 133.035, 103.058, 4.742, -139.298] deg; TCP offset x=-9.5 y=-328 z=105 mm, rx=1.2092 ry=-1.2092 rz=1.2092 rad
      MoveJ speed 60 deg/s, acceleration 80 deg/s^2 (useActiveTCP=true optimoveEnabled=false optiMoveSpeed=0.3 optiMoveAcceleration=0.09) feature=Base
        Waypoint Waypoint_13: TCP in base x=-820.615 y=235.067 z=-600.712 mm, rx=2.789 ry=-0.3984 rz=-1.1799 rad; joints [-36.349, -28.171, 124.415, -140.933, -100.235, -24.393] deg
      MoveL speed 250 mm/s, acceleration 1200 mm/s^2 (useActiveTCP=true optimoveEnabled=false optiMoveSpeed=0.3 optiMoveAcceleration=0.09) feature=Base
        Waypoint Waypoint_14: TCP in base x=-933.006 y=247.304 z=-556.073 mm, rx=2.8803 ry=-0.0661 rz=-1.2302 rad; joints [-29.557, -31.673, 118.683, -136.217, -107.709, -21.437] deg
      MoveJ speed 60 deg/s, acceleration 80 deg/s^2 (useActiveTCP=true optimoveEnabled=false optiMoveSpeed=0.3 optiMoveAcceleration=0.09) feature=Base
        Waypoint Waypoint_15: TCP in base x=-1155.523 y=247.304 z=-556.073 mm, rx=0.1075 ry=2.332 rz=-0.0118 rad; joints [-20.182, -12.844, 81.619, -201.64, -80.424, -192.34] deg
      'end of approach'
      SuppressedNode
        MoveL speed 250 mm/s, acceleration 1200 mm/s^2 (useActiveTCP=true optimoveEnabled=false optiMoveSpeed=0.3 optiMoveAcceleration=0.09) feature=Base
          Waypoint Waypoint_18: TCP in base x=-939.675 y=242.159 z=-688.931 mm, rx=0.1858 ry=2.4403 rz=-0.0331 rad; joints [-25.871, -6.691, 96.723, -229.022, -77.473, -192.661] deg; TCP offset x=4.51 y=-328 z=105 mm, rx=1.2092 ry=-1.2092 rz=1.2092 rad
          Waypoint Waypoint_19: TCP in base x=-939.675 y=242.159 z=-719.896 mm, rx=0.1858 ry=2.4403 rz=-0.0331 rad; joints [-25.872, -4.62, 94.895, -229.263, -77.472, -192.663] deg
      SuppressedNode
        Wait Sleep waitTime=2
      SuppressedNode
        MoveP speed 10 mm/s, acceleration 1200 mm/s^2 (blendRadius=0.025 useActiveTCP=true optimoveEnabled=false optiMoveSpeed=0.3 optiMoveAcceleration=0.09) feature=Base
          CircleMove (OrientationMode=FIXED)
            Waypoint ViaPoint_5: TCP in base x=-907.205 y=264.785 z=-719.9 mm, rx=1.8738 ry=1.7594 rz=-0.6531 rad; joints [-28.993, -7.691, 102.75, -211.731, -134.382, -127.614] deg
            Waypoint EndPoint_3: TCP in base x=-881.393 y=236.092 z=-719.9 mm, rx=-2.9216 ry=0.2235 rz=1.0597 rad; joints [-28.315, -21.001, 113.308, -133.575, -104.432, -14.143] deg
          CircleMove (OrientationMode=FIXED)
            Waypoint ViaPoint_6: TCP in base x=-912.548 y=210.58 z=-719.9 mm, rx=-1.7177 ry=1.9091 rz=0.6478 rad; joints [-24.877, -16.344, 111.718, -164.775, -43.133, 60.968] deg
            Waypoint Waypoint_19: TCP in base x=-939.675 y=242.159 z=-719.896 mm, rx=0.1858 ry=2.4403 rz=-0.0331 rad; joints [-25.872, -4.62, 94.895, -229.263, -77.472, -192.663] deg
          CircleMove (OrientationMode=FIXED)
            Waypoint ViaPoint_5: TCP in base x=-907.205 y=264.785 z=-719.9 mm, rx=1.8738 ry=1.7594 rz=-0.6531 rad; joints [-28.993, -7.691, 102.75, -211.731, -134.382, -127.614] deg
            Waypoint EndPoint_3: TCP in base x=-881.393 y=236.092 z=-719.9 mm, rx=-2.9216 ry=0.2235 rz=1.0597 rad; joints [-28.315, -21.001, 113.308, -133.575, -104.432, -14.143] deg
  MoveL speed 250 mm/s, acceleration 1200 mm/s^2 (useActiveTCP=true optimoveEnabled=false optiMoveSpeed=0.3 optiMoveAcceleration=0.09) feature=Base
    Waypoint Waypoint_21: TCP in base x=-970.523 y=290.955 z=-552.096 mm, rx=2.8078 ry=0.1074 rz=-1.2042 rad; joints [-31.638, -31.143, 114.281, -134.947, -112.801, 329.628] deg; TCP offset x=-9.5 y=-328 z=105 mm, rx=1.2092 ry=-1.2092 rz=1.2092 rad
  MoveJ speed 60 deg/s, acceleration 80 deg/s^2 (useActiveTCP=true optimoveEnabled=false optiMoveSpeed=0.3 optiMoveAcceleration=0.09) feature=Base
    Waypoint Waypoint_20: TCP in base x=-1155.523 y=247.304 z=-556.073 mm, rx=0.1075 ry=2.332 rz=-0.0118 rad; joints [-20.182, -12.844, 81.619, -201.64, -80.424, -192.34] deg
SubProgram extrude_knife3 (keepSynchronizedWithDisk=false) programFile=/programs/extrude_knife3.urp
  Folder pre program stuff
    Set NoAction tcp=pretend_welder
    ek_sp := get_actual_tcp_pose()
    MoveL speed 5 mm/s, acceleration 1200 mm/s^2 (useActiveTCP=true optimoveEnabled=false optiMoveSpeed=0.3 optiMoveAcceleration=0.09) feature=Base
      Waypoint Variable (Variable): variable=ek_sp
    SuppressedNode
      Script file /programs/analyze_touchpoints.script
        | # this file creates the function for analyzing touchpoints
        | # define pi
        | pi = 3.1415926535
        | # initialize a lift column extension needed of 0.0
        | global liftcolumnzneeded = 0.0
        | 
        | # this is the main entry point for calculations.
        | # it takes in the 5 points, analyzes the shape of the box, and then calculates path points and returns them
        | # specifically for Down, Over, then Around (DOtA)
        | # specifically for right-sided boxes (vertical weld on right side of edge)
        | def main_calculate_right(p11, p12, p21, p22, p3, p13, p23, chamferover):
        |     struct1 = analyze_touchpoints_only(p11, p12, p21, p22, p3)
        |     list1 = analyze_vertical_touchpoints(p11, p12, p13, p21, p22, p23, p3)
        |     struct2 = calculate_DOtA_points_right(struct1, list1, chamferover)
        |     validity = check_validity_right(struct1, struct2)
        |     return struct2
        | end
        | 
        | # this is the main entry point for calculations.
        | # it takes in the 5 points, analyzes the shape of the box, and then calculates path points and returns them
        | # specifically for Down, Over, then Around (DOtA)
        | # specifically for left-sided boxes (vertical weld on left side of edge)
        | def main_calculate_left(p11, p12, p21, p22, p3, p13, p23, chamferover):
        |     struct1 = analyze_touchpoints_only(p11, p12, p21, p22, p3)
        |     list1 = analyze_vertical_touchpoints(p11, p12, p13, p21, p22, p23, p3)
        |     struct2 = calculate_DOtA_points_left(struct1, list1, chamferover)
        |     validity = check_validity_left(struct1, struct2)
        |     return struct2
        | end
        | 
        | # this is the main entry point for calculations, for Floor Corner Extended.
        | # it takes in the 7 touchpoints, analyzes the shape of the box.
        | # takes in the user defined point for the top of the weld (tcp_pose_top) and then calculates path points
        | # loopingly tries to calculate the extension along the sidewall that fulfills get_inverse_kin_has_solution() and provides the farthest extension possible
        | # returns the pathpoints
        | # specifically for Down, Over, then Around (DOtA)
        | # specifically for right-sided boxes (vertical weld on right side of edge)
        | def main_calculate_right_extended(p11, p12, p21, p22, p3, p13, p23, chamferover, chamferup, tcp_pose_top):
        |     struct1 = analyze_touchpoints_only(p11, p12, p21, p22, p3)
        |     list1 = analyze_vertical_touchpoints(p11, p12, p13, p21, p22, p23, p3)
        |     struct2 = calculate_DOtA_points_right_extended(struct1, list1, chamferover, chamferup, tcp_pose_top)
        |     struct3 = check_validity_right(struct1, struct2)
        |     return struct3
        | end
        | 
        | # this is the main entry point for calculations, for Floor Corner Extended.
        | # it takes in the 7 touchpoints, analyzes the shape of the box.
        | # takes in the user defined point for the top of the weld (tcp_pose_top) and then calculates path points
        | # loopingly tries to calculate the extension along the sidewall that fulfills get_inverse_kin_has_solution() and provides the farthest extension possible
        | # returns the pathpoints
        | # specifically for Down, Over, then Around (DOtA)
        | # specifically for left-sided boxes (vertical weld on left side of edge)
        | def main_calculate_left_extended(p11, p12, p21, p22, p3, p13, p23, chamferover, chamferup, tcp_pose_top):
        |     struct1 = analyze_touchpoints_only(p11, p12, p21, p22, p3)
        |     list1 = analyze_vertical_touchpoints(p11, p12, p13, p21, p22, p23, p3)
        |     struct2 = calculate_DOtA_points_left_extended(struct1, list1, chamferover, chamferup, tcp_pose_top)
        |     struct3 = check_validity_left(struct1, struct2)
        |     return struct3
        | end
        | 
        | # it takes 5 arguments as points
        | # it returns a struct containing: (pointintersect, pointapproach1, pointapproach2, point1, point2, point3, point4, point5, pointreturn1, heading1, heading2, heading3, path2r1, path2r2, path2l1, path2l2)
        | # specifically for Around then Up (AtU)
        | def analyze_touchpoints(p11, p12, p21, p22, p3):
        |   # FIND THE INTERSECTION
        |   # comment get the z
        |   zcoord=p3[2]
        | 
        |   # get the raw points from the first line
        |   l1p1x=p11[0]
        |   l1p1y=p11[1]
        |   l1p2x=p12[0]
        |   l1p2y=p12[1]
        | 
        |   # equate the first line in 2d space
        |   ml1 = (l1p2y-l1p1y) / (l1p2x-l1p1x)
        | 
        |   # b = y - mx
        |   bl1 = l1p1y - ml1 * l1p1x
        | 
        |   # get the raw points from the second line
        |   l2p1x=p21[0]
        |   l2p1y=p21[1]
        |   l2p2x=p22[0]
        |   l2p2y=p22[1]
        | 
        |   # equate the second line in 2d space
        |   ml2 = (l2p2y-l2p1y) / (l2p2x-l2p1x)
        | 
        |   # b = y - mx
        |   bl2 = l2p1y - ml2 * l2p1x
        | 
        | 
        |   # find the intersection of the two lines
        |   # m1x+b1 = m2x+b2
        |   # m1x - m2x = b2 - b1
        |   # x = (b2-b1) / (m1-m2)
        |   xintersect = (bl2-bl1) / (ml1-ml2)
        |   yintersect = ml1 * xintersect + bl1
        | 
        |   #FIND THE VECTORS
        |   #define a vector from the intersection to the second point on the first line
        |   l1delxfull = l1p2x - xintersect
        |   l1delyfull = l1p2y - yintersect
        | 
        |   l1delmag = sqrt(l1delxfull*l1delxfull + l1delyfull*l1delyfull)
        | 
        |   l1delxunit = l1delxfull / l1delmag
        |   l1delyunit = l1delyfull / l1delmag
        | 
        |   #define a vector from the intersection to the second point on the second line
        |   l2delxfull = l2p2x - xintersect
        |   l2delyfull = l2p2y - yintersect
        | 
        |   l2delmag = sqrt(l2delxfull*l2delxfull + l2delyfull*l2delyfull)
        | 
        |   l2delxunit = l2delxfull / l2delmag
        |   l2delyunit = l2delyfull / l2delmag
        | 
        |   # FIND THE FOUR POINTS ON THE LINES
        |   # find locations 8 inches away from  intersect point
        |   # CONST
        |   welddistance = 8
        |   roundoverdistance = 0.05
        |   zup = .375
        |   # inches
        |   wd = welddistance * 25.4 / 1000
        |   rod = roundoverdistance * 25.4 / 1000
        |   zup = zup * 25.4 / 1000
        | 
        |   # now we have the unit vector. extend the weld distance from the intersection
        |   x = xintersect + l1delxunit * wd
        |   y = yintersect + l1delyunit * wd
        |   z = zcoord + zup
        | 
        |   point1 = p[x,y,z,1.570796,0,0] # dummy orientation for now
        | 
        |   x = xintersect + l1delxunit * rod
        |   y = yintersect + l1delyunit * rod
        | 
        |   point2 = p[x,y,z,1.570796,0,0]
        | 
        |   # now we have the unit vector. extend the weld distance from the intersection
        |   x = xintersect + l2delxunit * wd
        |   y = yintersect + l2delyunit * wd
        | 
        |   point5 = p[x,y,z,0,-1.570796,0]
        | 
        |   x = xintersect + l2delxunit * rod
        |   y = yintersect + l2delyunit * rod
        | 
        |   point4 = p[x,y,z,0,-1.570796,0]
        | 
        |   #DEFINE APPROACH POINTS
        |   pointintersect = p[xintersect,yintersect,zcoord,0,0,0]
        |   pointapproach1 = p[xintersect+0.1,yintersect+0.1,z,1.570796,0,0]
        |   pointapproach2 = p[point1[0], point1[1]+0.1, point1[2], point1[3], point1[4], point1[5]]
        |   pointreturn1 = p[point5[0]+0.1, point5[1], point5[2], point5[3], point5[4], point5[5]]
        | 
        |   #FIND HEADINGS
        |   #for each heading, find the angle of the line with respect to the pos x axis. then add/subtract 90 degrees because you want to be perpendicular to that
        |   headingvector1 = convert_uv_to_heading(l1delxunit, l1delyunit)
        |   headingvector2 = convert_uv_to_heading(l2delxunit, l2delyunit)
        |   # find halfway heading
        |   heading2 = (headingvector1 + headingvector2)/2
        |   # find headings that the robot should face while traveling, perpendicular to the vectors of the sides of the box
        |   heading1 = headingvector1 + pi/2
        |   heading3 = headingvector2 - pi/2
        | 
        |   #FIND POINT 3
        |   #see if we have to / can find point 3
        |   findpoint3 = True
        |   if roundoverdistance == 0:
        |     findpoint3 = False
        |   end
        |   if findpoint3:
        |     # i need to find the point3 such that the arc from p2 to p3 to p4 is tangent to p1-p2 and p4-p5. making this a smooth path will be good
        |     # the direction of movement is from pointintersect in the direction of heading2
        |     # how much movement though? this will depend on whether it is actually a 90 degree angle or not.
        |     # first, find the perpendicular lines through points 2 and 4
        |     perp2 = find_perpendicular_line(ml1, point2[0], point2[1])
        |     perp4 = find_perpendicular_line(ml2, point4[0], point4[1])
        |     # next, find the intersection of those two lines
        |     perpintersect = find_intersection(perp2[0], perp2[1], perp4[0], perp4[1])
        |     radiusofcircle = distance_between(perpintersect[0], perpintersect[1], 0, point2[0], point2[1], 0)
        |     # find a vector the direction of heading2
        |     uvx = cos(heading2)
        |     uvy = sin(heading2)
        |     # compute point3. pass in negative radius because the direction is into the tank but we want to move from the intersection out to the rounded edge
        |     point3coords = add_vectordistance_to_point(perpintersect[0], perpintersect[1], z, uvx, uvy, 0, -1 * radiusofcircle)
        |     point3 = p[point3coords[0], point3coords[1], point3coords[2], 0, 0, 0]
        |   end
        | 
        |   #APPLY ACTUAL RXRYRZ TO POINTS
        |   # convert the headings to rxryrz and insert those values into the relevant points
        |   rxryrz = convert_heading_to_axang(heading1)
        |   rx = rxryrz[0]
        |   ry = rxryrz[1]
        |   rz = rxryrz[2]
        |   pointapproach1 = p[pointapproach1[0], pointapproach1[1], pointapproach1[2], rx, ry, rz]
        |   pointapproach2 = p[pointapproach2[0], pointapproach2[1], pointapproach2[2], rx, ry, rz]
        |   point1 = p[point1[0], point1[1], point1[2], rx, ry, rz]
        |   point2 = p[point2[0], point2[1], point2[2], rx, ry, rz]
        |   rxryrz = convert_heading_to_axang(heading2)
        |   rx = rxryrz[0]
        |   ry = rxryrz[1]
        |   rz = rxryrz[2]
        |   if findpoint3:
        |     point3 = p[point3[0], point3[1], point3[2], rx, ry, rz]
        |   else:
        |     point3 = point2
        |   end
        |   rxryrz = convert_heading_to_axang(heading3)
        |   rx = rxryrz[0]
        |   ry = rxryrz[1]
        |   rz = rxryrz[2]
        |   point4 = p[point4[0], point4[1], point4[2], rx, ry, rz]
        |   point5 = p[point5[0], point5[1], point5[2], rx, ry, rz]
        |   pointreturn1 = p[pointreturn1[0], pointreturn1[1], pointreturn1[2], rx, ry, rz]
        | 
        |   #find path2 (the part that goes up)
        |   four_vertical_points = find_vertical_points(pointintersect, l1delxunit, l1delyunit, l2delxunit, l2delyunit, zup, wd, heading1, heading3)
        |   path2r1 = four_vertical_points[0]
        |   path2r2 = four_vertical_points[1]
        |   path2l1 = four_vertical_points[2]
        |   path2l2 = four_vertical_points[3]
        | 
        |   #RETURN STRUCT
        |   ret = struct(pointintersect=pointintersect, pointapproach1=pointapproach1, pointapproach2=pointapproach2, point1=point1, point2=point2, point3=point3, point4=point4, point5=point5, pointreturn1=pointreturn1, heading1=heading1, heading2=heading2, heading3=heading3, path2r1=path2r1, path2r2=path2r2, path2l1=path2l1, path2l2=path2l2)
        |   return ret
        | end
        | 
        | # it takes 5 arguments as points
        | # it returns a struct containing: (pointintersect, heading1, heading2, heading3, l1delxunit, l1delyunit, l2delxunit, l2delyunit)
        | def analyze_touchpoints_only(p11, p12, p21, p22, p3):
        |   # FIND THE INTERSECTION
        |   # comment get the z
        |   zcoord=p3[2]
        | 
        |   # get the raw points from the first line
        |   l1p1x=p11[0]
        |   l1p1y=p11[1]
        |   l1p2x=p12[0]
        |   l1p2y=p12[1]
        | 
        |   # equate the first line in 2d space
        |   ml1 = (l1p2y-l1p1y) / (l1p2x-l1p1x)
        | 
        |   # b = y - mx
        |   bl1 = l1p1y - ml1 * l1p1x
        | 
        |   # get the raw points from the second line
        |   l2p1x=p21[0]
        |   l2p1y=p21[1]
        |   l2p2x=p22[0]
        |   l2p2y=p22[1]
        | 
        |   # equate the second line in 2d space
        |   ml2 = (l2p2y-l2p1y) / (l2p2x-l2p1x)
        | 
        |   # b = y - mx
        |   bl2 = l2p1y - ml2 * l2p1x
        | 
        | 
        |   # find the intersection of the two lines
        |   # m1x+b1 = m2x+b2
        |   # m1x - m2x = b2 - b1
        |   # x = (b2-b1) / (m1-m2)
        |   xintersect = (bl2-bl1) / (ml1-ml2)
        |   yintersect = ml1 * xintersect + bl1
        | 
        |   pointintersect = p[xintersect,yintersect,zcoord,0,0,0]
        | 
        |   #FIND THE VECTORS
        |   #define a vector from the intersection to the second point on the first line
        |   l1delxfull = l1p2x - xintersect
        |   l1delyfull = l1p2y - yintersect
        | 
        |   l1delmag = sqrt(l1delxfull*l1delxfull + l1delyfull*l1delyfull)
        | 
        |   l1delxunit = l1delxfull / l1delmag
        |   l1delyunit = l1delyfull / l1delmag
        | 
        |   #define a vector from the intersection to the second point on the second line
        |   l2delxfull = l2p2x - xintersect
        |   l2delyfull = l2p2y - yintersect
        | 
        |   l2delmag = sqrt(l2delxfull*l2delxfull + l2delyfull*l2delyfull)
        | 
        |   l2delxunit = l2delxfull / l2delmag
        |   l2delyunit = l2delyfull / l2delmag
        | 
        |   #FIND HEADINGS
        |   #for each heading, find the angle of the line with respect to the pos x axis. then add/subtract 90 degrees because you want to be perpendicular to that
        |   headingvector1 = convert_uv_to_heading(l1delxunit, l1delyunit)
        |   headingvector2 = convert_uv_to_heading(l2delxunit, l2delyunit)
        |   # find halfway heading
        |   heading2 = (headingvector1 + headingvector2)/2
        |   # find headings that the robot should face while traveling, perpendicular to the vectors of the sides of the box
        |   heading1 = headingvector1 + pi/2
        |   heading3 = headingvector2 - pi/2
        | 
        |   #RETURN STRUCT
        |   ret = struct(pointintersect=pointintersect, heading1=heading1, heading2=heading2, heading3=heading3, l1delxunit=l1delxunit, l1delyunit=l1delyunit, l2delxunit=l2delxunit, l2delyunit=l2delyunit)
        |   return ret
        | end
        | 
        | # given a struct from analyze_touchpoints_only(), calculate the points
        | # for right, for non-extended
        | def calculate_DOtA_points_right(struct1, listleans, chamferover):
        |     # get the stuff from the struct
        |     pointintersect = struct1[0]
        |     heading1 = struct1[1]
        |     heading2 = struct1[2]
        |     heading3 = struct1[3]
        |     l1delxunit = struct1[4]
        |     l1delyunit = struct1[5]
        |     l2delxunit = struct1[6]
        |     l2delyunit = struct1[7]
        | 
        |     # FIND THE POINTS ON THE LINES OF THE FIRST TURN PATH
        |     # find locations 8 inches away from  intersect point
        |     # CONST
        |     welddistance1 = 8 # vertical weld distance
        |     welddistance2 = 6 # first path second leg
        |     welddistance3 = 8 # second path second leg
        |     zup = .375
        |     # inches
        |     wd1 = welddistance1 * 25.4 / 1000
        |     wd2 = welddistance2 * 25.4 / 1000
        |     wd3 = welddistance3 * 25.4 / 1000
        |     zup = zup * 25.4 / 1000
        |     chamferovermm =  chamferover * 25.4 / 1000
        | 
        |     x = pointintersect[0] + l1delxunit * chamferovermm
        |     y = pointintersect[1] + l1delyunit * chamferovermm
        |     z = pointintersect[2] + zup
        | 
        |     #apply actual rxryrz to points
        |     # convert the headings to rxryrz and insert those values into the relevant points
        |     rxryrz = convert_heading_to_axang_preheatdown(heading1)
        |     rx = rxryrz[0]
        |     ry = rxryrz[1]
        |     rz = rxryrz[2]
        | 
        |     point1 = p[x + wd1*listleans[0], y + wd1*listleans[1], z + wd1, rx, ry, rz] # add in the listleans factor to follow the face of the box as we move up
        |     point2 = p[x, y, z, rx, ry, rz]
        | 
        |     # convert the headings to rxryrz and insert those values into the relevant points
        |     rxryrz = convert_heading_to_axang_ccw(heading1)
        |     rx = rxryrz[0]
        |     ry = rxryrz[1]
        |     rz = rxryrz[2]
        | 
        |     point4 = p[x, y, z, rx, ry, rz]
        |     x = x + l1delxunit * wd2
        |     y = y + l1delyunit * wd2
        |     point5 = p[x, y, z, rx, ry, rz]
        | 
        |     # FIND THE POINTS ON THE LINES OF THE SECOND AROUND PATH
        |     roundoverdistance = 0.05
        |     rod = roundoverdistance * 25.4 / 1000
        | 
        |     # now we have the unit vector. extend the weld distance from the intersection
        |     x = pointintersect[0] + l1delxunit * chamferovermm
        |     y = pointintersect[1] + l1delyunit * chamferovermm
        |     # convert the headings to rxryrz and insert those values into the relevant points
        |     rxryrz = convert_heading_to_axang(heading1)
        |     rx = rxryrz[0]
        |     ry = rxryrz[1]
        |     rz = rxryrz[2]
        |     point_1 = p[x, y, z, rx, ry, rz]
        | 
        |     x = pointintersect[0] + l1delxunit * rod
        |     y = pointintersect[1] + l1delyunit * rod
        |     point_2 = p[x, y, z, rx, ry, rz]
        | 
        |     # now we have the unit vector. extend the weld distance from the intersection
        |     x = pointintersect[0] + l2delxunit * wd3
        |     y = pointintersect[1] + l2delyunit * wd3
        |     # convert the headings to rxryrz and insert those values into the relevant points
        |     rxryrz = convert_heading_to_axang(heading3)
        |     rx = rxryrz[0]
        |     ry = rxryrz[1]
        |     rz = rxryrz[2]
        |     point_5 = p[x, y, z, rx, ry, rz]
        | 
        |     x = pointintersect[0] + l2delxunit * rod
        |     y = pointintersect[1] + l2delyunit * rod
        |     point_4 = p[x, y, z, rx, ry, rz]
        | 
        |     #FIND POINT 3
        |     # by calling analyze_touchpoints()
        |     atret = analyze_touchpoints(point_2, point_1, point_4, point_5, pointintersect)
        |     point_3 = atret[5]
        | 
        | 
        |     struct2 = struct(point1=point1, point2=point2, point4=point4, point5=point5, point_1=point_1, point_2=point_2, point_3=point_3, point_4=point_4, point_5=point_5)
        |     return struct2
        | end
        | 
        | # given a struct from analyze_touchpoints_only(), calculate the points
        | # for left, for non-extended
        | def calculate_DOtA_points_left(struct1, listleans, chamferover):
        |     # get the stuff from the struct
        |     pointintersect = struct1[0]
        |     heading1 = struct1[1]
        |     heading2 = struct1[2]
        |     heading3 = struct1[3]
        |     l1delxunit = struct1[4]
        |     l1delyunit = struct1[5]
        |     l2delxunit = struct1[6]
        |     l2delyunit = struct1[7]
        | 
        |     # FIND THE POINTS ON THE LINES OF THE FIRST TURN PATH
        |     # find locations 8 inches away from  intersect point
        |     # CONST
        |     welddistance1 = 8 # vertical weld distance
        |     welddistance2 = 6 # first path second leg
        |     welddistance3 = 8 # second path second leg
        |     zup = .375
        |     # inches
        |     wd1 = welddistance1 * 25.4 / 1000
        |     wd2 = welddistance2 * 25.4 / 1000
        |     wd3 = welddistance3 * 25.4 / 1000
        |     zup = zup * 25.4 / 1000
        |     chamferovermm =  chamferover * 25.4 / 1000
        | 
        |     x = pointintersect[0] + l2delxunit * chamferovermm
        |     y = pointintersect[1] + l2delyunit * chamferovermm
        |     z = pointintersect[2] + zup
        | 
        |     #apply actual rxryrz to points
        |     # convert the headings to rxryrz and insert those values into the relevant points
        |     rxryrz = convert_heading_to_axang_preheatdown(heading3)
        |     rx = rxryrz[0]
        |     ry = rxryrz[1]
        |     rz = rxryrz[2]
        | 
        |     point1 = p[x + wd1*listleans[0], y + wd1*listleans[1], z + wd1, rx, ry, rz]
        |     point2 = p[x, y, z, rx, ry, rz]
        | 
        |     # convert the headings to rxryrz and insert those values into the relevant points
        |     rxryrz = convert_heading_to_axang(heading3)
        |     rx = rxryrz[0]
        |     ry = rxryrz[1]
        |     rz = rxryrz[2]
        | 
        |     point4 = p[x, y, z, rx, ry, rz]
        |     x = x + l2delxunit * wd2
        |     y = y + l2delyunit * wd2
        |     point5 = p[x, y, z, rx, ry, rz]
        | 
        |     # FIND THE POINTS ON THE LINES OF THE SECOND AROUND PATH
        |     roundoverdistance = 0.05
        |     rod = roundoverdistance * 25.4 / 1000
        | 
        |     # now we have the unit vector. extend the weld distance from the intersection
        |     x = pointintersect[0] + l2delxunit * chamferovermm
        |     y = pointintersect[1] + l2delyunit * chamferovermm
        |     # convert the headings to rxryrz and insert those values into the relevant points
        |     rxryrz = convert_heading_to_axang_ccw(heading3)
        |     rx = rxryrz[0]
        |     ry = rxryrz[1]
        |     rz = rxryrz[2]
        |     point_1 = p[x, y, z, rx, ry, rz]
        | 
        |     x = pointintersect[0] + l2delxunit * rod
        |     y = pointintersect[1] + l2delyunit * rod
        |     point_2 = p[x, y, z, rx, ry, rz]
        | 
        |     # now we have the unit vector. extend the weld distance from the intersection
        |     x = pointintersect[0] + l1delxunit * wd3
        |     y = pointintersect[1] + l1delyunit * wd3
        |     # convert the headings to rxryrz and insert those values into the relevant points
        |     rxryrz = convert_heading_to_axang_ccw(heading1)
        |     rx = rxryrz[0]
        |     ry = rxryrz[1]
        |     rz = rxryrz[2]
        |     point_5 = p[x, y, z, rx, ry, rz]
        | 
        |     x = pointintersect[0] + l1delxunit * rod
        |     y = pointintersect[1] + l1delyunit * rod
        |     point_4 = p[x, y, z, rx, ry, rz]
        | 
        |     #FIND POINT 3
        |     # by calling analyze_touchpoints()
        |     atret = analyze_touchpoints(point_2, point_1, point_4, point_5, pointintersect)
        |     point_3 = atret[5]
        |     #point 3 will not have the correct rxryrz though because now the gun needs to be face up.
        |     rxryrz = convert_heading_to_axang_ccw(heading2)
        |     rx = rxryrz[0]
        |     ry = rxryrz[1]
        |     rz = rxryrz[2]
        |     point_3 = p[point_3[0], point_3[1], point_3[2], rx, ry, rz]
        | 
        |     struct2 = struct(point1=point1, point2=point2, point4=point4, point5=point5, point_1=point_1, point_2=point_2, point_3=point_3, point_4=point_4, point_5=point_5)
        |     return struct2
        | end
        | 
        | # given a struct from analyze_touchpoints_only(), calculate the points
        | # for right, for extended
        | def calculate_DOtA_points_right_extended(struct1, listleans, chamferover, chamferup, tcp_pose_top):
        |     # get the stuff from the struct
        |     pointintersect = struct1[0]
        |     heading1 = struct1[1]
        |     heading2 = struct1[2]
        |     heading3 = struct1[3]
        |     l1delxunit = struct1[4]
        |     l1delyunit = struct1[5]
        |     l2delxunit = struct1[6]
        |     l2delyunit = struct1[7]
        | 
        |     # FIND THE POINTS ON THE LINES OF THE FIRST TURN PATH
        |     # find locations 8 inches away from  intersect point
        |     # CONST
        |     # welddistance1 = 8 # vertical weld distance
        |     welddistance2 = 6 # first path second leg
        |     welddistance3 = 8 # second path second leg
        | 
        |     # inches
        |     # wd1 = welddistance1 * 25.4 / 1000
        |     wd2 = welddistance2 * 25.4 / 1000
        |     wd3 = welddistance3 * 25.4 / 1000
        |     zup = chamferup * 25.4 / 1000
        |     chamferovermm =  chamferover * 25.4 / 1000
        | 
        |     # weld distance is the distance that it will weld. this will make it start at the z height that the user specified
        |     wd1 = tcp_pose_top[2] - pointintersect[2] - zup
        | 
        |     x = pointintersect[0] + l1delxunit * chamferovermm
        |     y = pointintersect[1] + l1delyunit * chamferovermm
        |     z = pointintersect[2] + zup
        | 
        |     #apply actual rxryrz to points
        |     # convert the headings to rxryrz and insert those values into the relevant points
        |     rxryrz = convert_heading_to_axang_preheatdown(heading1)
        |     rx = rxryrz[0]
        |     ry = rxryrz[1]
        |     rz = rxryrz[2]
        | 
        |     point1 = p[x + wd1*listleans[0], y + wd1*listleans[1], z + wd1, rx, ry, rz] # add in the listleans factor to follow the face of the box as we move up
        |     point2 = p[x, y, z, rx, ry, rz]
        | 
        |     # convert the headings to rxryrz and insert those values into the relevant points
        |     rxryrz = convert_heading_to_axang_ccw(heading1)
        |     rx = rxryrz[0]
        |     ry = rxryrz[1]
        |     rz = rxryrz[2]
        | 
        |     point4 = p[x, y, z, rx, ry, rz]
        |     x = x + l1delxunit * wd2
        |     y = y + l1delyunit * wd2
        |     point5 = p[x, y, z, rx, ry, rz]
        | 
        |     # FIND THE POINTS ON THE LINES OF THE SECOND AROUND PATH
        |     roundoverdistance = 0.05
        |     rod = roundoverdistance * 25.4 / 1000
        | 
        |     # now we have the unit vector. extend the weld distance from the intersection
        |     x = pointintersect[0] + l1delxunit * chamferovermm
        |     y = pointintersect[1] + l1delyunit * chamferovermm
        |     # convert the headings to rxryrz and insert those values into the relevant points
        |     rxryrz = convert_heading_to_axang(heading1)
        |     rx = rxryrz[0]
        |     ry = rxryrz[1]
        |     rz = rxryrz[2]
        |     point_1 = p[x, y, z, rx, ry, rz]
        | 
        |     x = pointintersect[0] + l1delxunit * rod
        |     y = pointintersect[1] + l1delyunit * rod
        |     point_2 = p[x, y, z, rx, ry, rz]
        | 
        |     # convert the headings to rxryrz and insert those values into the relevant points
        |     rxryrz = convert_heading_to_axang(heading3)
        |     rx = rxryrz[0]
        |     ry = rxryrz[1]
        |     rz = rxryrz[2]
        | 
        |     x = pointintersect[0] + l2delxunit * rod
        |     y = pointintersect[1] + l2delyunit * rod
        |     point_4 = p[x, y, z, rx, ry, rz]
        | 
        |     # now we have the unit vector. extend the weld distance from the intersection
        |     x = pointintersect[0] + l2delxunit * wd3
        |     y = pointintersect[1] + l2delyunit * wd3
        |     point_5 = p[x, y, z, rx, ry, rz]
        | 
        |     #FIND POINT 3
        |     # by calling analyze_touchpoints()
        |     atret = analyze_touchpoints(point_2, point_1, point_4, point_5, pointintersect)
        |     point_3 = atret[5]
        | 
        | 
        |     struct2 = struct(point1=point1, point2=point2, point4=point4, point5=point5, point_1=point_1, point_2=point_2, point_3=point_3, point_4=point_4, point_5=point_5)
        |     return struct2
        | end
        | 
        | # given a struct from analyze_touchpoints_only(), calculate the points
        | # for left, for extended
        | def calculate_DOtA_points_left_extended(struct1, listleans, chamferover, chamferup, tcp_pose_top):
        |     # get the stuff from the struct
        |     pointintersect = struct1[0]
        |     heading1 = struct1[1]
        |     heading2 = struct1[2]
        |     heading3 = struct1[3]
        |     l1delxunit = struct1[4]
        |     l1delyunit = struct1[5]
        |     l2delxunit = struct1[6]
        |     l2delyunit = struct1[7]
        | 
        |     # FIND THE POINTS ON THE LINES OF THE FIRST TURN PATH
        |     # find locations 8 inches away from  intersect point
        |     # CONST
        |     # welddistance1 = 8 # vertical weld distance
        |     welddistance2 = 6 # first path second leg
        |     welddistance3 = 8 # second path second leg
        | 
        |     # inches
        |     # wd1 = welddistance1 * 25.4 / 1000
        |     wd2 = welddistance2 * 25.4 / 1000
        |     wd3 = welddistance3 * 25.4 / 1000
        |     zup = chamferup * 25.4 / 1000
        |     chamferovermm =  chamferover * 25.4 / 1000
        | 
        |     # weld distance is the distance that it will weld. this will make it start at the z height that the user specified
        |     wd1 = tcp_pose_top[2] - pointintersect[2] - zup
        | 
        |     x = pointintersect[0] + l2delxunit * chamferovermm
        |     y = pointintersect[1] + l2delyunit * chamferovermm
        |     z = pointintersect[2] + zup
        | 
        |     #apply actual rxryrz to points
        |     # convert the headings to rxryrz and insert those values into the relevant points
        |     rxryrz = convert_heading_to_axang_preheatdown(heading3)
        |     rx = rxryrz[0]
        |     ry = rxryrz[1]
        |     rz = rxryrz[2]
        | 
        |     point1 = p[x + wd1*listleans[0], y + wd1*listleans[1], z + wd1, rx, ry, rz]
        |     point2 = p[x, y, z, rx, ry, rz]
        | 
        |     # convert the headings to rxryrz and insert those values into the relevant points
        |     rxryrz = convert_heading_to_axang(heading3)
        |     rx = rxryrz[0]
        |     ry = rxryrz[1]
        |     rz = rxryrz[2]
        | 
        |     point4 = p[x, y, z, rx, ry, rz]
        |     x = x + l2delxunit * wd2
        |     y = y + l2delyunit * wd2
        |     point5 = p[x, y, z, rx, ry, rz]
        | 
        |     # FIND THE POINTS ON THE LINES OF THE SECOND AROUND PATH
        |     roundoverdistance = 0.05
        |     rod = roundoverdistance * 25.4 / 1000
        | 
        |     # now we have the unit vector. extend the weld distance from the intersection
        |     x = pointintersect[0] + l2delxunit * chamferovermm
        |     y = pointintersect[1] + l2delyunit * chamferovermm
        |     # convert the headings to rxryrz and insert those values into the relevant points
        |     rxryrz = convert_heading_to_axang_ccw(heading3)
        |     rx = rxryrz[0]
        |     ry = rxryrz[1]
        |     rz = rxryrz[2]
        |     point_1 = p[x, y, z, rx, ry, rz]
        | 
        |     x = pointintersect[0] + l2delxunit * rod
        |     y = pointintersect[1] + l2delyunit * rod
        |     point_2 = p[x, y, z, rx, ry, rz]
        | 
        |     # convert the headings to rxryrz and insert those values into the relevant points
        |     rxryrz = convert_heading_to_axang_ccw(heading1)
        |     rx = rxryrz[0]
        |     ry = rxryrz[1]
        |     rz = rxryrz[2]
        | 
        |     x = pointintersect[0] + l1delxunit * rod
        |     y = pointintersect[1] + l1delyunit * rod
        |     point_4 = p[x, y, z, rx, ry, rz]
        | 
        |     # now we have the unit vector. extend the weld distance from the intersection
        |     x = pointintersect[0] + l1delxunit * wd3
        |     y = pointintersect[1] + l1delyunit * wd3
        |     point_5 = p[x, y, z, rx, ry, rz]
        | 
        |     #FIND POINT 3
        |     # by calling analyze_touchpoints()
        |     atret = analyze_touchpoints(point_2, point_1, point_4, point_5, pointintersect)
        |     point_3 = atret[5]
        |     #point 3 will not have the correct rxryrz though because now the gun needs to be face up
        |     rxryrz = convert_heading_to_axang_ccw(heading2)
        |     rx = rxryrz[0]
        |     ry = rxryrz[1]
        |     rz = rxryrz[2]
        |     point_3 = p[point_3[0], point_3[1], point_3[2], rx, ry, rz]
        | 
        |     struct2 = struct(point1=point1, point2=point2, point4=point4, point5=point5, point_1=point_1, point_2=point_2, point_3=point_3, point_4=point_4, point_5=point_5)
        |     return struct2
        | end
        | 
        | # this function analyzes the vertical points
        | # calculates the slope of the edge in question
        | # specifically, for each inch up in the z direction, what is the change in x and change in y direction
        | # returns a list of [nx, ny]
        | def analyze_vertical_touchpoints(p11, p12, p13, p21, p22, p23, p3):
        |     # first, find the equations of the planes from the 6 points
        |     plane1 = findplane(p11, p12, p13)
        |     plane2 = findplane(p21, p22, p23)
        |     # Find the Direction Vector of the Line: The direction vector d of the line of intersection can be found by taking the cross product of the normal vectors of each plane (a, b, and c)
        |     nx = plane1[1]*plane2[2] - plane1[2]*plane2[1]
        |     ny = plane1[2]*plane2[0] - plane1[0]*plane2[2]
        |     nz = plane1[0]*plane2[1] - plane1[1]*plane2[0]
        |     # normalize the vector so the z length is 1
        |     multiplier = 1 / nz
        |     nx = nx * multiplier
        |     ny = ny * multiplier
        |     nz = nz * multiplier # should become equal to 1
        |     ret = [nx, ny]
        |     return ret
        | end
        | 
        | # given 3 points, this finds the plane and its equation
        | # rereturns ax + by + cz + d = 0 in a list of [a, b, c, d]
        | def findplane(p11, p12, p13):
        |     # extract coordinates
        |     x1 = p11[0]
        |     y1 = p11[1]
        |     z1 = p11[2]
        |     x2 = p12[0]
        |     y2 = p12[1]
        |     z2 = p12[2]
        |     x3 = p13[0]
        |     y3 = p13[1]
        |     z3 = p13[2]
        |     # create vectors from the points
        |     v1x = x2-x1
        |     v1y = y2-y1
        |     v1z = z2-z1
        |     v2x = x3-x1
        |     v2y = y3-y1
        |     v2z = z3-z1
        |     #calculate the normal vector using the cross product
        |     nx = v1y*v2z - v1z*v2y # i component
        |     ny = v1z*v2x - v1x*v2z # j component
        |     nz = v1x*v2y - v1y*v2x # k component
        |     # calculate d in the plane equation
        |     d = -1 * (nx*x1 + ny*y1 + nz*z1)
        |     ret = [nx, ny, nz, d]
        |     return ret
        | end
        | 
        | # given a heading, (ccw from +x axis), find the mx+b slope
        | # fails if exactly vertical
        | def get_slope_from_heading(heading):
        |     return tan(heading)
        | end
        | 
        | 
        | 
        | # this function finds the points (and rxryrz) of the 2 points (start and end) of vertical weld section
        | def find_vertical_points(pointintersect, l1delxunit, l1delyunit, l2delxunit, l2delyunit, offset, wd, heading1, heading3):
        | 
        |   # find right side stuff
        |   # find the point in 3d space that is .375 up and .375 over
        |   x = pointintersect[0] + l1delxunit * offset
        |   y = pointintersect[1] + l1delyunit * offset
        |   z = pointintersect[2] + offset
        |   # find rxryrz
        |   rxryrz = convert_heading_to_axang_preheatup(heading1)
        |   rx = rxryrz[0]
        |   ry = rxryrz[1]
        |   rz = rxryrz[2]
        |   path2r1 = p[x, y, z, rx, ry, rz]
        |   path2r2 = p[x, y, z + wd, rx, ry, rz]
        | 
        |   # find left side
        |   # find the point in 3d space that is .375 up and .375 over
        |   x = pointintersect[0] + l2delxunit * offset
        |   y = pointintersect[1] + l2delyunit * offset
        |   z = pointintersect[2] + offset
        |   # find rxryrz
        |   rxryrz = convert_heading_to_axang_preheatup(heading3)
        |   rx = rxryrz[0]
        |   ry = rxryrz[1]
        |   rz = rxryrz[2]
        |   path2l1 = p[x, y, z, rx, ry, rz]
        |   path2l2 = p[x, y, z + wd, rx, ry, rz]
        | 
        |   ret = struct(path2r1=path2r1, path2r2=path2r2, path2l1=path2l1, path2l2=path2l2)
        |   return ret
        | end
        | 
        | # this function converts a unit vector to its heading angle ccw from x+ axis
        | # takes uvx and uvy
        | # returns heading in radians
        | def convert_uv_to_heading(uvx, uvy):
        |   baseang = atan(uvy/uvx)
        |   if uvx < 0:
        |     ang = baseang + pi
        |   elif uvy < 0:
        |     ang = baseang + pi * 2
        |   else:
        |     ang = baseang
        |   end
        |   return ang
        | end
        | 
        | # this function finds the equation of a line, perpendicular to a given line, and going through a given point
        | # takes 3 arguments: m (the original line's slope), x (point's x coord), y (point's y coord). the b of the original line is not needed
        | # returns a list of [m,b] (the slope and intercept of the new line)
        | def find_perpendicular_line(origm, x, y):
        |   m = (1/origm) * -1
        |   b = y - m*x
        |   ret = [m, b]
        |   return ret
        | end
        | 
        | # this function finds the intersection point between two lines in the xy plane
        | # takes 4 arguments: m1, b1, m2, b2
        | # returns a list of [x,y] (the point of intersection)
        | def find_intersection(m1, b1, m2, b2):
        |   # m1x+b1 = m2x+b2
        |   # m1x - m2x = b2 - b1
        |   # x = (b2-b1) / (m1-m2)
        |   x = (b2-b1) / (m1-m2)
        |   y = m1 * x + b1
        |   ret = [x, y]
        |   return ret
        | end
        | 
        | # this function finds the distance between 2 points in 3d space
        | # it takes 6 arguments: x1, y1, z1, x2, y2, z2
        | # it returns a distance
        | def distance_between(x1, y1, z1, x2, y2, z2):
        |   distsquared = (x2-x1)*(x2-x1)+(y2-y1)*(y2-y1)+(z2-z1)*(z2-z1)
        |   dist = sqrt(distsquared)
        |   return dist
        | end
        | 
        | # this function takes a point, a unit vector, and a distance, and adds the distance to the point in the direction of the unit vector (3d space)
        | # it returns a point as a list of coordinates
        | def add_vectordistance_to_point(xi, yi, zi, uvx, uvy, uvz, delta):
        |   xf = xi + uvx * delta
        |   yf = yi + uvy * delta
        |   zf = zi + uvz * delta
        |   ret = [xf, yf, zf]
        |   return ret
        | end
        | 
        | # this function converts a heading (ccw radians from the positive x axis) into rxryrz to be put into a point p[]
        | # this will point the gun in this heading with the bottom side of the gun facing up.
        | # the values used in this program were calculated by doing rotation matrix math in the file on WI-CALVINB10 C. Documents. Theory for converting rotations into axis angle representations
        | def convert_heading_to_axang(heading):
        |  axisxraw = -1 * sin(heading)
        |  axisyraw = cos(heading) + 1
        |  axiszraw = sin(heading)
        | 
        |  magnitude = sqrt(axisxraw*axisxraw + axisyraw*axisyraw + axiszraw*axiszraw)
        | 
        |  axisxunit = axisxraw / magnitude
        |  axisyunit = axisyraw / magnitude
        |  axiszunit = axiszraw / magnitude
        | 
        |  angle = acos( (cos(heading) - 1) / 2 )
        | 
        |  rxout = axisxunit * angle
        |  ryout = axisyunit * angle
        |  rzout = axiszunit * angle
        | 
        |  return [rxout, ryout, rzout]
        | end
        | 
        | # this function converts a heading (ccw radians from the positive x axis) into rxryrz to be put into a point p[]
        | # this will point the gun in this heading with the preheat side of the gun tip facing up. Used for welding in a vertical path.
        | # the values used in this program were calculated by doing rotation matrix math in the file on WI-CALVINB10 C. Documents. Theory for converting rotations into axis angle representations
        | def convert_heading_to_axang_preheatup(heading):
        |  axisxraw = -sin(heading) + 1
        |  axisyraw = cos(heading)
        |  axiszraw = cos(heading)
        | 
        |  magnitude = sqrt(axisxraw*axisxraw + axisyraw*axisyraw + axiszraw*axiszraw)
        | 
        |  axisxunit = axisxraw / magnitude
        |  axisyunit = axisyraw / magnitude
        |  axiszunit = axiszraw / magnitude
        | 
        |  angle = acos( (-sin(heading) - 1) / 2 )
        | 
        |  rxout = axisxunit * angle
        |  ryout = axisyunit * angle
        |  rzout = axiszunit * angle
        | 
        |  return [rxout, ryout, rzout]
        | end
        | 
        | # this function converts a heading (ccw radians from the positive x axis) into rxryrz to be put into a point p[]
        | # this will point the gun in this heading with the preheat side of the gun tip facing down. Used for welding in a vertical path downwards.
        | # the values used in this program were calculated by doing rotation matrix math in the file on WI-CALVINB10 C. Documents. Theory for converting rotations into axis angle representations
        | def convert_heading_to_axang_preheatdown(heading):
        |  axisxraw = -sin(heading) - 1
        |  axisyraw = cos(heading)
        |  axiszraw = -cos(heading)
        | 
        |  magnitude = sqrt(axisxraw*axisxraw + axisyraw*axisyraw + axiszraw*axiszraw)
        | 
        |  axisxunit = axisxraw / magnitude
        |  axisyunit = axisyraw / magnitude
        |  axiszunit = axiszraw / magnitude
        | 
        |  angle = acos( (sin(heading) - 1) / 2 )
        | 
        |  rxout = axisxunit * angle
        |  ryout = axisyunit * angle
        |  rzout = axiszunit * angle
        | 
        |  return [rxout, ryout, rzout]
        | end
        | 
        | # this function converts a heading (ccw radians from the positive x axis) into rxryrz to be put into a point p[]
        | # this will point the gun in this heading with the preheat side of the gun tip facing right. Used for welding counterclockwise around the box.
        | # the values used in this program were calculated by doing rotation matrix math in the file on WI-CALVINB10 C. Documents. Theory for converting rotations into axis angle representations
        | def convert_heading_to_axang_ccw(heading):
        |  axisxraw = -sin(heading)
        |  axisyraw = cos(heading) - 1
        |  axiszraw = -sin(heading)
        | 
        |  magnitude = sqrt(axisxraw*axisxraw + axisyraw*axisyraw + axiszraw*axiszraw)
        | 
        |  axisxunit = axisxraw / magnitude
        |  axisyunit = axisyraw / magnitude
        |  axiszunit = axiszraw / magnitude
        | 
        |  angle = acos( (-cos(heading) - 1) / 2 )
        | 
        |  rxout = axisxunit * angle
        |  ryout = axisyunit * angle
        |  rzout = axiszunit * angle
        | 
        |  return [rxout, ryout, rzout]
        | end
        | 
        | # this function takes two rotation matrices, and multiplies them together, returning one matrix.
        | # all matrices are in the form of a list.
        | # all matrix values have constant values (no variables)
        | def multiply_matrix(matrix1, matrix2):
        |     # retrieve values
        |     a11 = matrix1[0]
        |     a12 = matrix1[1]
        |     a13 = matrix1[2]
        |     a21 = matrix1[3]
        |     a22 = matrix1[4]
        |     a23 = matrix1[5]
        |     a31 = matrix1[6]
        |     a32 = matrix1[7]
        |     a33 = matrix1[8]
        |     b11 = matrix2[0]
        |     b12 = matrix2[1]
        |     b13 = matrix2[2]
        |     b21 = matrix2[3]
        |     b22 = matrix2[4]
        |     b23 = matrix2[5]
        |     b31 = matrix2[6]
        |     b32 = matrix2[7]
        |     b33 = matrix2[8]
        |     #calculate c values
        |     c11 = a11*b11 + a12*b21 + a13*b31
        |     c12 = a11*b12 + a12*b22 + a13*b32
        |     c13 = a11*b13 + a12*b23 + a13*b33
        |     c21 = a21*b11 + a22*b21 + a23*b31
        |     c22 = a21*b12 + a22*b22 + a23*b32
        |     c23 = a21*b13 + a22*b23 + a23*b33
        |     c31 = a31*b11 + a32*b21 + a33*b31
        |     c32 = a31*b12 + a32*b22 + a33*b32
        |     c33 = a31*b13 + a32*b23 + a33*b33
        |     # return resulting matrix
        |     ret = [c11, c12, c13, c21, c22, c23, c31, c32, c33]
        |     return ret
        | end
        | 
        | # this function converts a matrix to axis angle representations
        | # this matrix is usually a resulting matrix (result of matrix multiplication) in normal use, given as a list
        | # returns a list of [rx,ry,rz]
        | def convert_matrix_to_axang(matrix1):
        |     # retrieve values
        |     a11 = matrix1[0]
        |     a12 = matrix1[1]
        |     a13 = matrix1[2]
        |     a21 = matrix1[3]
        |     a22 = matrix1[4]
        |     a23 = matrix1[5]
        |     a31 = matrix1[6]
        |     a32 = matrix1[7]
        |     a33 = matrix1[8]
        | 
        |     # First Half: find the angle
        |     # find the trace
        |     # using the formula: trace = a11 + a22 + a33
        |     trace = a11 + a22 + a33
        |     # find the angle using the formula: trace(matrix) = 1 + 2 cos(angle)
        |     angle = acos((trace - 1.0)/2.0)
        | 
        |     # Second Half: calculate the rotation axis
        |     axisxraw = a32 - a23
        |     axisyraw = a13 - a31
        |     axiszraw = a21 - a12
        |     # normalize axis
        |     magnitude = sqrt(axisxraw*axisxraw + axisyraw*axisyraw + axiszraw*axiszraw)
        |     axisxunit = axisxraw / magnitude
        |     axisyunit = axisyraw / magnitude
        |     axiszunit = axiszraw / magnitude
        | 
        |     # combine axis and angle into rxryrz representation
        |     rxout = axisxunit * angle
        |     ryout = axisyunit * angle
        |     rzout = axiszunit * angle
        |     return [rxout, ryout, rzout]
        | end
        | 
        | # this function takes a rotation and calculates the corresponding rotation matrix
        | # input is (axis, direction, angle in radians)
        | # example is ("x", 1, pi/6) = a 30 degree turn around the x axis in the positive direction (right hand rule)
        | # returns a matrix (a list of 9 values)
        | def get_rotation_matrix_from_description(axis, direction, angle):
        |     # get the angle
        |     a = angle * direction
        |     # get the axis
        |     if axis == "x" or axis == "X":
        |         matrix = [1, 0, 0, 0, cos(a), -1 * sin(a), 0, sin(a), cos(a)]
        |         return matrix
        |     end
        |     if axis == "y" or axis == "Y":
        |         matrix = [cos(a), 0, sin(a), 0, 1, 0, -1*sin(a), 0, cos(a)]
        |         return matrix
        |     end
        |     if axis == "z" or axis == "Z":
        |         matrix = [cos(a), -1*sin(a), 0, sin(a), cos(a), 0, 0, 0, 1]
        |         return matrix
        |     end
        |     # bad
        |     popuptext = "Error in get_rotation_matrix_from_description. "
        |     # infinite loop
        |     while 1==1:
        |       popup(popuptext, title="Code Error",blocking=True)
        |     end
        | end
        | 
        | # this function is for getting the points along the path of the corner homing 45
        | # point0 is the point where they touched
        | def get_corner_homing_45_pathpoints(point0, pointtop = p[0,0,0,0,0,0]):
        |   p0x = point0[0]
        |   p0y = point0[1]
        |   p0z = point0[2]
        |   p0rx = point0[3]
        |   p0ry = point0[4]
        |   p0rz = point0[5]
        | 
        |   #constants
        |   #distances of how far away from point the touchpoints are
        |   d0 = 0.10 # how far from the box to retreat and approach
        |   d1 = 0.03 # first distance from init point
        |   d2 = 0.15 # second distance from init point
        |   d3 = 0.125 #vertical distance from first point
        |   sqrt2 = 0.707106781 # 1/sqrt(2) , the inverse of the sqrt(2)
        | 
        |   ph1 = p[p0x + d0, p0y, p0z + d1, p0rx, p0ry, p0rz] #approach point for turn
        | 
        |   ph2 = p[p0x+d0-d0*0.5-sqrt2*d1, p0y+d0*0.5+sqrt2*d1, p0z+d1, 1.446, -0.8, -0.733]
        |   ph3 = p[p0x+d0-d0*0.5-sqrt2*d2, p0y+d0*0.5+sqrt2*d2, p0z+d1, 1.446, -0.8, -0.733]
        |   ph4 = p[p0x+d0-d0*0.5-sqrt2*d1, p0y-d0*0.5-sqrt2*d1, p0z+d1, 0.626, -1.993, -1.813]
        |   ph5 = p[p0x+d0-d0*0.5-sqrt2*d2, p0y-d0*0.5-sqrt2*d2, p0z+d1, 0.626, -1.993, -1.813]
        | 
        |   # go back to ph1
        |   ph6 = p[p0x + d0, p0y, p0z -0.05, 0, 0, 0] # approach point for under turn
        |   # moveL from ph1 to ph6
        |   ph7 = p[p0x-d1, p0y, p0z-0.05, 0, 0, 0]
        | 
        |   # add the vertical touch points
        |   if pointtop[2] == 0:
        |     ph2up = p[ph2[0], ph2[1], ph2[2]+d3, ph2[3], ph2[4], ph2[5]]
        |     ph4up = p[ph4[0], ph4[1], ph4[2]+d3, ph4[3], ph4[4], ph4[5]]
        |   elif pointtop[2] > p0z + 0.914: # 0.914m = 36 inches
        |     ph2up = p[ph2[0], ph2[1], p0z + 0.914, ph2[3], ph2[4], ph2[5]]
        |     ph4up = p[ph4[0], ph4[1], p0z + 0.914, ph4[3], ph4[4], ph4[5]]
        |   else:
        |     ph2up = p[ph2[0], ph2[1], pointtop[2], ph2[3], ph2[4], ph2[5]]
        |     ph4up = p[ph4[0], ph4[1], pointtop[2], ph4[3], ph4[4], ph4[5]]
        |   end
        |   ret = struct(ph1=ph1, ph2=ph2, ph3=ph3, ph4=ph4, ph5=ph5, ph6=ph6, ph7=ph7, ph2up=ph2up, ph4up=ph4up)
        |   is_robot_at_reachable_spot(point0, ret)
        |   return ret
        | end
        | 
